KUKA KRL program: EPS_2_251825_SA25_A_20260116064101.src

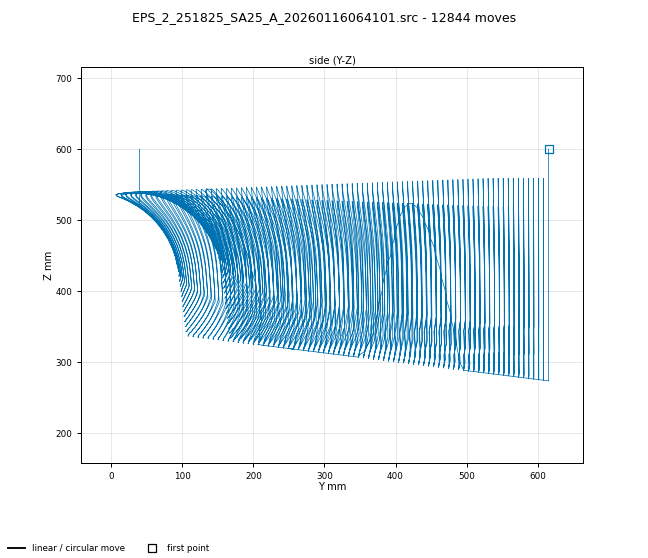
[picture p0: tool path of EPS_2_251825_SA25_A_20260116064101.src, 12844 of 12846 moves have a stored position in this frame; points joined in program order, loops and branches not executed]
&ACCESS RVP
&REL 4
&COMMENT QRS 19112012
&PARAM EDITMASK = *
DEF PART()
EXT BAS (BAS_COMMAND :IN,REAL :IN )
INT I
BAS (#INITMOV,0 )

;KUKA QRS Post kuka4.cps  Date:22-06-2017 !

File_ID=2984

QRS_PRE_INIT()

;Init var - Until changes are made in qrs_pre_init
Outlet_Square_prg=0
Inlet_1_Square_prg=0
Inlet_2_Square_prg=0
Inlet_3_Square_prg=0
Inlet_4_Square_prg=0
Inlet_5_Square_prg=0

Outlet_1={X 0.000, Y 535.490, Z 458.500, B 0.000, E1 0.000 }
Inlet_1={X 0.000, Y 538.340, Z 418.500, B 0.000, E1 170.000 }
Outlet_1_type=201
Inlet_1_type=201
;QRS#1=Sidecore dimensions
;QRS#2=200-8" PVC SDR 35
;QRS#3=200-8" PVC SDR 35
;QRS#4=
;QRS#5=
;QRS#6=
;QRS#7=
;QRS#8=
;QRS#9=12-08 PSX
;QRS#10=12-08 PSX
;QRS#11=
;QRS#12=
;QRS#13=
;QRS#14=
;QRS#15=
;QRS#16=1220x127x838 2,75'
;QRS#17=EPS Height
;QRS#18=559
;QRS#19=*
;QRS#20= UPDATED VERSION 22-06-2017
;QRS#21=*
Outlet_Square=0100
Inlet_1_Square=0100
Inlet_2_Square=0
Inlet_3_Square=0
Inlet_4_Square=0
Inlet_5_Square=0
Mill_Square=1
Outlet_Square_Prg=204
Inlet_1_Square_prg=204

QRS_INIT()

$ADVANCE=5

; T1
PTP {E1 173.614,E2 173.614}
PTP {X 0,Y 615.487,A -85,B 0,C 180,E1 173.614,E2 173.614,E3 0,E4 0,E5 0,E6 0}
QRS_SPEED_INIT()
LIN {X 0,Y 615.487,Z 600,A -85,B 0,C 180,E1 173.614,E2 173.614,E3 0,E4 0,E5 0,E6 0} C_VEL
LIN {X 0,Y 615.487,Z 283.875,A -85,B 0,C 180,E1 173.614,E2 173.614} C_VEL
LIN {X 0,Y 615.487,Z 275.693,A -85,B 0,C 180,E1 173.614,E2 173.614} C_VEL
LIN {X 0,Y 615.476,Z 273.693,A -85,B 0,C 180,E1 173.428,E2 173.428} C_VEL
LIN {X 0,Y 615.49,Z 273.68,A -85,B 0,C 180,E1 170.801,E2 170.801} C_VEL
LIN {X 0,Y 615.476,Z 273.688,A -85,B 0,C 180,E1 168.139,E2 168.139} C_VEL
LIN {X 0,Y 615.493,Z 273.698,A -85,B 0,C 180,E1 165.451,E2 165.451} C_VEL
LIN {X 0,Y 615.476,Z 273.685,A -85,B 0,C 180,E1 162.729,E2 162.729} C_VEL
LIN {X 0,Y 615.478,Z 273.686,A -85,B 0,C 180,E1 159.967,E2 159.967} C_VEL
LIN {X 0,Y 615.49,Z 273.698,A -85,B 0,C 180,E1 157.156,E2 157.156} C_VEL
LIN {X 0,Y 615.488,Z 273.681,A -85,B 0,C 180,E1 154.284,E2 154.284} C_VEL
LIN {X 0,Y 615.477,Z 273.689,A -85,B 0,C 180,E1 151.551,E2 151.551} C_VEL
LIN {X 0,Y 615.482,Z 273.7,A -85,B 0,C 180,E1 148.914,E2 148.914} C_VEL
LIN {X 0,Y 615.49,Z 273.68,A -85,B 0,C 180,E1 145.978,E2 145.978} C_VEL
LIN {X 0,Y 615.483,Z 273.694,A -85,B 0,C 180,E1 143.063,E2 143.063} C_VEL
LIN {X 0,Y 615.472,Z 273.69,A -85,B 0,C 180,E1 140.249,E2 140.249} C_VEL
LIN {X 0,Y 615.494,Z 273.679,A -85,B 0,C 180,E1 137.647,E2 137.647} C_VEL
LIN {X 0,Y 615.478,Z 273.692,A -85,B 0,C 180,E1 134.93,E2 134.93} C_VEL
LIN {X 0,Y 615.473,Z 273.692,A -85,B 0,C 180,E1 132.079,E2 132.079} C_VEL
LIN {X 0,Y 615.472,Z 273.686,A -85,B 0,C 180,E1 129.751,E2 129.751} C_VEL
LIN {X 0,Y 615.481,Z 273.685,A -85,B 0,C 180,E1 126.936,E2 126.936} C_VEL
LIN {X 0,Y 615.482,Z 273.696,A -85,B 0,C 180,E1 124.022,E2 124.022} C_VEL
LIN {X 0,Y 615.471,Z 273.691,A -85,B 0,C 180,E1 121.686,E2 121.686} C_VEL
LIN {X 0,Y 615.471,Z 273.686,A -85,B 0,C 180,E1 119.407,E2 119.407} C_VEL
LIN {X 0,Y 615.481,Z 273.787,A -85,B 0,C 180,E1 118.606,E2 118.606} C_VEL
LIN {X 0,Y 615.47,Z 289.754,A -85,B 0,C 180,E1 115.898,E2 115.898} C_VEL
LIN {X 0,Y 615.442,Z 304.793,A -85,B 0,C 180,E1 113.38,E2 113.38} C_VEL
LIN {X 0,Y 615.49,Z 308.179,A -85,B 0,C 180,E1 112.813,E2 112.813} C_VEL
LIN {X 0,Y 615.422,Z 414.922,A -85,B 0,C 180,E1 111.544,E2 111.544} C_VEL
LIN {X 0,Y 615.433,Z 427.931,A -85,B 0,C 180,E1 111.258,E2 111.258} C_VEL
LIN {X 0,Y 615.473,Z 440.076,A -85,B 0,C 180,E1 110.862,E2 110.862} C_VEL
LIN {X 0,Y 615.47,Z 451.61,A -85,B 0,C 180,E1 110.359,E2 110.359} C_VEL
LIN {X 0,Y 615.466,Z 462.135,A -85,B 0,C 180,E1 109.773,E2 109.773} C_VEL
LIN {X 0,Y 615.497,Z 473.243,A -85,B 0,C 180,E1 108.991,E2 108.991} C_VEL
LIN {X 0,Y 615.499,Z 481.455,A -85,B 0,C 180,E1 108.282,E2 108.282} C_VEL
LIN {X 0,Y 615.497,Z 489.66,A -85,B 0,C 180,E1 107.442,E2 107.442} C_VEL
LIN {X 0,Y 615.496,Z 497.619,A -85,B 0,C 180,E1 106.433,E2 106.433} C_VEL
LIN {X 0,Y 615.495,Z 503.176,A -85,B 0,C 180,E1 105.565,E2 105.565} C_VEL
LIN {X 0,Y 615.497,Z 508.401,A -85,B 0,C 180,E1 104.549,E2 104.549} C_VEL
LIN {X 0,Y 615.496,Z 512.408,A -85,B 0,C 180,E1 103.537,E2 103.537} C_VEL
LIN {X 0,Y 615.494,Z 515.337,A -85,B 0,C 180,E1 102.53,E2 102.53} C_VEL
LIN {X 0,Y 615.496,Z 516.703,A -85,B 0,C 180,E1 101.861,E2 101.861} C_VEL
LIN {X 0,Y 615.496,Z 518.232,A -85,B 0,C 180,E1 100.527,E2 100.527} C_VEL
LIN {X 0,Y 615.496,Z 518.372,A -85,B 0,C 180,E1 99.862,E2 99.862} C_VEL
LIN {X 0,Y 615.496,Z 517.451,A -85,B 0,C 180,E1 98.537,E2 98.537} C_VEL
LIN {X 0,Y 615.494,Z 516.408,A -85,B 0,C 180,E1 97.876,E2 97.876} C_VEL
LIN {X 0,Y 615.495,Z 513.082,A -85,B 0,C 180,E1 96.583,E2 96.583} C_VEL
LIN {X 0,Y 615.496,Z 509.298,A -85,B 0,C 180,E1 95.57,E2 95.57} C_VEL
LIN {X 0,Y 615.498,Z 504.497,A -85,B 0,C 180,E1 94.585,E2 94.585} C_VEL
LIN {X 0,Y 615.491,Z 498.461,A -85,B 0,C 180,E1 93.601,E2 93.601} C_VEL
LIN {X 0,Y 615.498,Z 490.972,A -85,B 0,C 180,E1 92.618,E2 92.618} C_VEL
LIN {X 0,Y 615.497,Z 483.209,A -85,B 0,C 180,E1 91.8,E2 91.8} C_VEL
LIN {X 0,Y 615.5,Z 475.088,A -85,B 0,C 180,E1 91.064,E2 91.064} C_VEL
LIN {X 0,Y 615.493,Z 465.046,A -85,B 0,C 180,E1 90.327,E2 90.327} C_VEL
LIN {X 0,Y 615.486,Z 453.961,A -85,B 0,C 180,E1 89.673,E2 89.673} C_VEL
LIN {X 0,Y 615.491,Z 443.467,A -85,B 0,C 180,E1 89.183,E2 89.183} C_VEL
LIN {X 0,Y 615.461,Z 430.84,A -85,B 0,C 180,E1 88.733,E2 88.733} C_VEL
LIN {X 0,Y 615.462,Z 418.151,A -85,B 0,C 180,E1 88.426,E2 88.426} C_VEL
LIN {X 0,Y 615.475,Z 400.264,A -85,B 0,C 180,E1 88.18,E2 88.18} C_VEL
LIN {X 0,Y 615.467,Z 308.178,A -85,B 0,C 180,E1 87.096,E2 87.096} C_VEL
LIN {X 0,Y 615.429,Z 294.206,A -85,B 0,C 180,E1 84.759,E2 84.759} C_VEL
LIN {X 0,Y 615.432,Z 280.557,A -85,B 0,C 180,E1 82.454,E2 82.454} C_VEL
LIN {X 0,Y 615.438,Z 273.696,A -85,B 0,C 180,E1 81.256,E2 81.256} C_VEL
LIN {X 0,Y 615.418,Z 273.696,A -85,B 0,C 180,E1 78.806,E2 78.806} C_VEL
LIN {X 0,Y 615.42,Z 273.696,A -85,B 0,C 180,E1 76.798,E2 76.798} C_VEL
LIN {X 0,Y 615.42,Z 273.696,A -85,B 0,C 180,E1 74.773,E2 74.773} C_VEL
LIN {X 0,Y 615.424,Z 273.695,A -85,B 0,C 180,E1 72.728,E2 72.728} C_VEL
LIN {X 0,Y 615.424,Z 273.695,A -85,B 0,C 180,E1 70.661,E2 70.661} C_VEL
LIN {X 0,Y 615.425,Z 273.695,A -85,B 0,C 180,E1 68.567,E2 68.567} C_VEL
LIN {X 0,Y 615.423,Z 273.695,A -85,B 0,C 180,E1 66.442,E2 66.442} C_VEL
LIN {X 0,Y 615.425,Z 273.695,A -85,B 0,C 180,E1 64.282,E2 64.282} C_VEL
LIN {X 0,Y 615.428,Z 273.696,A -85,B 0,C 180,E1 62.083,E2 62.083} C_VEL
LIN {X 0,Y 615.492,Z 273.695,A -85,B 0,C 180,E1 59.081,E2 59.081} C_VEL
LIN {X 0,Y 615.448,Z 273.691,A -85,B 0,C 180,E1 56.471,E2 56.471} C_VEL
LIN {X 0,Y 615.434,Z 273.693,A -85,B 0,C 180,E1 54.173,E2 54.173} C_VEL
LIN {X 0,Y 615.432,Z 273.694,A -85,B 0,C 180,E1 51.929,E2 51.929} C_VEL
LIN {X 0,Y 615.452,Z 273.697,A -85,B 0,C 180,E1 49.392,E2 49.392} C_VEL
LIN {X 0,Y 615.497,Z 273.694,A -85,B 0,C 180,E1 46.757,E2 46.757} C_VEL
LIN {X 0,Y 615.447,Z 273.69,A -85,B 0,C 180,E1 43.995,E2 43.995} C_VEL
LIN {X 0,Y 615.439,Z 273.694,A -85,B 0,C 180,E1 41.478,E2 41.478} C_VEL
LIN {X 0,Y 615.473,Z 273.699,A -85,B 0,C 180,E1 38.905,E2 38.905} C_VEL
LIN {X 0,Y 615.495,Z 273.692,A -85,B 0,C 180,E1 36.424,E2 36.424} C_VEL
LIN {X 0,Y 615.485,Z 273.685,A -85,B 0,C 180,E1 34.022,E2 34.022} C_VEL
LIN {X 0,Y 615.458,Z 273.688,A -85,B 0,C 180,E1 31.687,E2 31.687} C_VEL
LIN {X 0,Y 615.446,Z 273.69,A -85,B 0,C 180,E1 29.408,E2 29.408} C_VEL
LIN {X 0,Y 615.446,Z 273.693,A -85,B 0,C 180,E1 27.04,E2 27.04} C_VEL
LIN {X 0,Y 615.492,Z 273.699,A -85,B 0,C 180,E1 24.272,E2 24.272} C_VEL
LIN {X 0,Y 615.467,Z 273.686,A -85,B 0,C 180,E1 21.433,E2 21.433} C_VEL
LIN {X 0,Y 615.466,Z 273.686,A -85,B 0,C 180,E1 19.339,E2 19.339} C_VEL
LIN {X 0,Y 615.463,Z 273.686,A -85,B 0,C 180,E1 17.271,E2 17.271} C_VEL
LIN {X 0,Y 615.469,Z 273.685,A -85,B 0,C 180,E1 15.226,E2 15.226} C_VEL
LIN {X 0,Y 615.473,Z 273.685,A -85,B 0,C 180,E1 13.201,E2 13.201} C_VEL
LIN {X 0,Y 615.454,Z 273.692,A -85,B 0,C 180,E1 10.527,E2 10.527} C_VEL
LIN {X 0,Y 615.487,Z 273.702,A -85,B 0,C 180,E1 7.876,E2 7.876} C_VEL
LIN {X 0,Y 615.491,Z 273.684,A -85,B 0,C 180,E1 5.241,E2 5.241} C_VEL
LIN {X 0,Y 615.46,Z 273.687,A -85,B 0,C 180,E1 2.618,E2 2.618} C_VEL
LIN {X 0,Y 615.469,Z 273.695,A -85,B 0,C 180,E1 0,E2 0} C_VEL
LIN {X 0,Y 615.489,Z 273.693,A -85,B 0,C 180,E1 -2.618,E2 -2.618} C_VEL
LIN {X 0,Y 615.487,Z 273.682,A -85,B 0,C 180,E1 -5.241,E2 -5.241} C_VEL
LIN {X 0,Y 615.461,Z 273.689,A -85,B 0,C 180,E1 -7.876,E2 -7.876} C_VEL
LIN {X 0,Y 615.485,Z 273.701,A -85,B 0,C 180,E1 -10.527,E2 -10.527} C_VEL
LIN {X 0,Y 615.487,Z 273.686,A -85,B 0,C 180,E1 -13.201,E2 -13.201} C_VEL
LIN {X 0,Y 615.469,Z 273.685,A -85,B 0,C 180,E1 -15.906,E2 -15.906} C_VEL
LIN {X 0,Y 615.48,Z 273.698,A -85,B 0,C 180,E1 -18.646,E2 -18.646} C_VEL
LIN {X 0,Y 615.48,Z 273.687,A -85,B 0,C 180,E1 -21.432,E2 -21.432} C_VEL
LIN {X 0,Y 615.468,Z 273.687,A -85,B 0,C 180,E1 -24.273,E2 -24.273} C_VEL
LIN {X 0,Y 615.496,Z 273.701,A -85,B 0,C 180,E1 -27.049,E2 -27.049} C_VEL
LIN {X 0,Y 615.487,Z 273.683,A -85,B 0,C 180,E1 -29.797,E2 -29.797} C_VEL
LIN {X 0,Y 615.473,Z 273.686,A -85,B 0,C 180,E1 -32.459,E2 -32.459} C_VEL
LIN {X 0,Y 615.472,Z 273.691,A -85,B 0,C 180,E1 -34.816,E2 -34.816} C_VEL
LIN {X 0,Y 615.487,Z 273.7,A -85,B 0,C 180,E1 -37.242,E2 -37.242} C_VEL
LIN {X 0,Y 615.481,Z 273.684,A -85,B 0,C 180,E1 -40.09,E2 -40.09} C_VEL
LIN {X 0,Y 615.494,Z 273.679,A -85,B 0,C 180,E1 -42.353,E2 -42.353} C_VEL
LIN {X 0,Y 615.475,Z 273.69,A -85,B 0,C 180,E1 -45.07,E2 -45.07} C_VEL
LIN {X 0,Y 615.478,Z 273.693,A -85,B 0,C 180,E1 -47.921,E2 -47.921} C_VEL
LIN {X 0,Y 615.475,Z 273.687,A -85,B 0,C 180,E1 -50.25,E2 -50.25} C_VEL
LIN {X 0,Y 615.481,Z 273.685,A -85,B 0,C 180,E1 -53.065,E2 -53.065} C_VEL
LIN {X 0,Y 615.485,Z 273.697,A -85,B 0,C 180,E1 -55.979,E2 -55.979} C_VEL
LIN {X 0,Y 615.472,Z 273.691,A -85,B 0,C 180,E1 -58.315,E2 -58.315} C_VEL
LIN {X 0,Y 615.472,Z 273.687,A -85,B 0,C 180,E1 -60.594,E2 -60.594} C_VEL
LIN {X 0,Y 615.487,Z 273.681,A -85,B 0,C 180,E1 -62.956,E2 -62.956} C_VEL
LIN {X 0,Y 615.481,Z 273.692,A -85,B 0,C 180,E1 -65.728,E2 -65.728} C_VEL
LIN {X 0,Y 615.487,Z 273.756,A -85,B 0,C 180,E1 -67.438,E2 -67.438} C_VEL
LIN {X 0,Y 615.455,Z 293.696,A -85,B 0,C 180,E1 -70.141,E2 -70.141} C_VEL
LIN {X 0,Y 615.472,Z 313.082,A -85,B 0,C 180,E1 -72.73,E2 -72.73} C_VEL
LIN {X 0,Y 615.493,Z 334.92,A -85,B 0,C 180,E1 -75.607,E2 -75.607} C_VEL
LIN {X 0,Y 615.471,Z 346.472,A -85,B 0,C 180,E1 -77.114,E2 -77.114} C_VEL
LIN {X 0,Y 615.457,Z 454.866,A -85,B 0,C 180,E1 -78.411,E2 -78.411} C_VEL
LIN {X 0,Y 615.456,Z 467.368,A -85,B 0,C 180,E1 -78.682,E2 -78.682} C_VEL
LIN {X 0,Y 615.483,Z 480.688,A -85,B 0,C 180,E1 -79.116,E2 -79.116} C_VEL
LIN {X 0,Y 615.492,Z 492.486,A -85,B 0,C 180,E1 -79.64,E2 -79.64} C_VEL
LIN {X 0,Y 615.483,Z 504.003,A -85,B 0,C 180,E1 -80.304,E2 -80.304} C_VEL
LIN {X 0,Y 615.499,Z 514.347,A -85,B 0,C 180,E1 -81.05,E2 -81.05} C_VEL
LIN {X 0,Y 615.497,Z 522.696,A -85,B 0,C 180,E1 -81.795,E2 -81.795} C_VEL
LIN {X 0,Y 615.498,Z 530.61,A -85,B 0,C 180,E1 -82.62,E2 -82.62} C_VEL
LIN {X 0,Y 615.491,Z 538.207,A -85,B 0,C 180,E1 -83.608,E2 -83.608} C_VEL
LIN {X 0,Y 615.498,Z 545.207,A -85,B 0,C 180,E1 -84.759,E2 -84.759} C_VEL
LIN {X 0,Y 615.493,Z 549.853,A -85,B 0,C 180,E1 -85.744,E2 -85.744} C_VEL
LIN {X 0,Y 615.494,Z 553.4,A -85,B 0,C 180,E1 -86.727,E2 -86.727} C_VEL
LIN {X 0,Y 615.497,Z 555.234,A -85,B 0,C 180,E1 -87.383,E2 -87.383} C_VEL
LIN {X 0,Y 615.497,Z 556.609,A -85,B 0,C 180,E1 -88.037,E2 -88.037} C_VEL
LIN {X 0,Y 615.496,Z 558.174,A -85,B 0,C 180,E1 -89.346,E2 -89.346} C_VEL
LIN {X 0,Y 615.494,Z 558.389,A -85,B 0,C 180,E1 -90,E2 -90} C_VEL
LIN {X 0,Y 615.495,Z 557.58,A -85,B 0,C 180,E1 -91.309,E2 -91.309} C_VEL
LIN {X 0,Y 615.497,Z 556.608,A -85,B 0,C 180,E1 -91.963,E2 -91.963} C_VEL
LIN {X 0,Y 615.497,Z 555.232,A -85,B 0,C 180,E1 -92.618,E2 -92.618} C_VEL
LIN {X 0,Y 615.496,Z 552.348,A -85,B 0,C 180,E1 -93.601,E2 -93.601} C_VEL
LIN {X 0,Y 615.498,Z 548.44,A -85,B 0,C 180,E1 -94.585,E2 -94.585} C_VEL
LIN {X 0,Y 615.499,Z 543.403,A -85,B 0,C 180,E1 -95.57,E2 -95.57} C_VEL
LIN {X 0,Y 615.49,Z 536.913,A -85,B 0,C 180,E1 -96.578,E2 -96.578} C_VEL
LIN {X 0,Y 615.497,Z 529.131,A -85,B 0,C 180,E1 -97.546,E2 -97.546} C_VEL
LIN {X 0,Y 615.498,Z 519.255,A -85,B 0,C 180,E1 -98.537,E2 -98.537} C_VEL
LIN {X 0,Y 615.495,Z 508.863,A -85,B 0,C 180,E1 -99.365,E2 -99.365} C_VEL
LIN {X 0,Y 615.482,Z 498.572,A -85,B 0,C 180,E1 -100.029,E2 -100.029} C_VEL
LIN {X 0,Y 615.495,Z 487.133,A -85,B 0,C 180,E1 -100.616,E2 -100.616} C_VEL
LIN {X 0,Y 615.467,Z 475.354,A -85,B 0,C 180,E1 -101.078,E2 -101.078} C_VEL
LIN {X 0,Y 615.455,Z 462.238,A -85,B 0,C 180,E1 -101.444,E2 -101.444} C_VEL
LIN {X 0,Y 615.461,Z 448.933,A -85,B 0,C 180,E1 -101.674,E2 -101.674} C_VEL
LIN {X 0,Y 615.471,Z 346.467,A -85,B 0,C 180,E1 -102.887,E2 -102.887} C_VEL
LIN {X 0,Y 615.455,Z 325.989,A -85,B 0,C 180,E1 -105.566,E2 -105.566} C_VEL
LIN {X 0,Y 615.481,Z 305.474,A -85,B 0,C 180,E1 -108.281,E2 -108.281} C_VEL
LIN {X 0,Y 615.468,Z 283.343,A -85,B 0,C 180,E1 -111.257,E2 -111.257} C_VEL
LIN {X 0,Y 615.489,Z 273.682,A -85,B 0,C 180,E1 -112.594,E2 -112.594} C_VEL
LIN {X 0,Y 615.485,Z 273.681,A -85,B 0,C 180,E1 -114.992,E2 -114.992} C_VEL
LIN {X 0,Y 615.482,Z 273.698,A -85,B 0,C 180,E1 -117.915,E2 -117.915} C_VEL
LIN {X 0,Y 615.486,Z 273.682,A -85,B 0,C 180,E1 -120.92,E2 -120.92} C_VEL
LIN {X 0,Y 615.471,Z 273.686,A -85,B 0,C 180,E1 -123.531,E2 -123.531} C_VEL
LIN {X 0,Y 615.486,Z 273.699,A -85,B 0,C 180,E1 -126.425,E2 -126.425} C_VEL
LIN {X 0,Y 615.481,Z 273.685,A -85,B 0,C 180,E1 -129.061,E2 -129.061} C_VEL
LIN {X 0,Y 615.491,Z 273.68,A -85,B 0,C 180,E1 -131.473,E2 -131.473} C_VEL
LIN {X 0,Y 615.469,Z 273.692,A -85,B 0,C 180,E1 -134.151,E2 -134.151} C_VEL
LIN {X 0,Y 615.482,Z 273.693,A -85,B 0,C 180,E1 -136.953,E2 -136.953} C_VEL
LIN {X 0,Y 615.483,Z 273.684,A -85,B 0,C 180,E1 -139.393,E2 -139.393} C_VEL
LIN {X 0,Y 615.479,Z 273.683,A -85,B 0,C 180,E1 -141.989,E2 -141.989} C_VEL
LIN {X 0,Y 615.471,Z 273.69,A -85,B 0,C 180,E1 -144.383,E2 -144.383} C_VEL
LIN {X 0,Y 615.477,Z 273.697,A -85,B 0,C 180,E1 -146.763,E2 -146.763} C_VEL
LIN {X 0,Y 615.487,Z 273.701,A -85,B 0,C 180,E1 -149.08,E2 -149.08} C_VEL
LIN {X 0,Y 615.484,Z 273.681,A -85,B 0,C 180,E1 -152.085,E2 -152.085} C_VEL
LIN {X 0,Y 615.482,Z 273.696,A -85,B 0,C 180,E1 -155.008,E2 -155.008} C_VEL
LIN {X 0,Y 615.478,Z 273.687,A -85,B 0,C 180,E1 -157.863,E2 -157.863} C_VEL
LIN {X 0,Y 615.477,Z 273.684,A -85,B 0,C 180,E1 -160.662,E2 -160.662} C_VEL
LIN {X 0,Y 615.486,Z 273.7,A -85,B 0,C 180,E1 -163.568,E2 -163.568} C_VEL
LIN {X 0,Y 615.476,Z 273.688,A -85,B 0,C 180,E1 -166.125,E2 -166.125} C_VEL
LIN {X 0,Y 615.485,Z 273.681,A -85,B 0,C 180,E1 -168.807,E2 -168.807} C_VEL
LIN {X 0,Y 615.479,Z 273.694,A -85,B 0,C 180,E1 -171.463,E2 -171.463} C_VEL
LIN {X 0,Y 615.48,Z 273.694,A -85,B 0,C 180,E1 -174.101,E2 -174.101} C_VEL
LIN {X 0,Y 615.487,Z 273.681,A -85,B 0,C 180,E1 -176.727,E2 -176.727} C_VEL
LIN {X 0,Y 615.474,Z 273.686,A -85,B 0,C 180,E1 -179.346,E2 -179.346} C_VEL
LIN {X 0,Y 615.49,Z 273.698,A -85,B 0,C 180,E1 -181.963,E2 -181.963} C_VEL
LIN {X 0,Y 615.476,Z 273.69,A -85,B 0,C 180,E1 -184.585,E2 -184.585} C_VEL
LIN {X 0,Y 615.476,Z 273.693,A -85,B 0,C 180,E1 -186.572,E2 -186.572} C_VEL
LIN {X 0,Y 614.808,Z 273.83,A -85,B 0,C 180,E1 -187.118,E2 -187.118} C_VEL
LIN {X 0,Y 611.982,Z 274.253,A -85,B 0,C 180,E1 -188.004,E2 -188.004} C_VEL
LIN {X 0,Y 609.591,Z 274.559,A -85,B 0,C 180,E1 -188.717,E2 -188.717} C_VEL
LIN {X 0,Y 608.551,Z 274.675,A -85,B 0,C 180,E1 -189.267,E2 -189.267} C_VEL
LIN {X 0,Y 608.459,Z 274.686,A -85,B 0,C 180,E1 -189.453,E2 -189.453} C_VEL
LIN {X 0,Y 608.454,Z 274.691,A -85,B 0,C 180,E1 -192,E2 -192} C_VEL
LIN {X 0,Y 608.477,Z 274.69,A -85,B 0,C 180,E1 -194.72,E2 -194.72} C_VEL
LIN {X 0,Y 608.444,Z 274.687,A -85,B 0,C 180,E1 -197.477,E2 -197.477} C_VEL
LIN {X 0,Y 608.445,Z 274.687,A -85,B 0,C 180,E1 -199.571,E2 -199.571} C_VEL
LIN {X 0,Y 608.474,Z 274.689,A -85,B 0,C 180,E1 -202.405,E2 -202.405} C_VEL
LIN {X 0,Y 608.448,Z 274.694,A -85,B 0,C 180,E1 -204.571,E2 -204.571} C_VEL
LIN {X 0,Y 608.473,Z 274.689,A -85,B 0,C 180,E1 -207.207,E2 -207.207} C_VEL
LIN {X 0,Y 608.466,Z 274.685,A -85,B 0,C 180,E1 -209.972,E2 -209.972} C_VEL
LIN {X 0,Y 608.452,Z 274.695,A -85,B 0,C 180,E1 -212.88,E2 -212.88} C_VEL
LIN {X 0,Y 608.434,Z 274.697,A -85,B 0,C 180,E1 -215.278,E2 -215.278} C_VEL
LIN {X 0,Y 608.467,Z 274.687,A -85,B 0,C 180,E1 -217.746,E2 -217.746} C_VEL
LIN {X 0,Y 608.446,Z 274.687,A -85,B 0,C 180,E1 -220.329,E2 -220.329} C_VEL
LIN {X 0,Y 608.477,Z 274.694,A -85,B 0,C 180,E1 -223.31,E2 -223.31} C_VEL
LIN {X 0,Y 608.459,Z 274.687,A -85,B 0,C 180,E1 -226.13,E2 -226.13} C_VEL
LIN {X 0,Y 608.454,Z 274.687,A -85,B 0,C 180,E1 -228.824,E2 -228.824} C_VEL
LIN {X 0,Y 608.46,Z 274.695,A -85,B 0,C 180,E1 -231.761,E2 -231.761} C_VEL
LIN {X 0,Y 608.444,Z 274.694,A -85,B 0,C 180,E1 -233.955,E2 -233.955} C_VEL
LIN {X 0,Y 608.442,Z 274.69,A -85,B 0,C 180,E1 -236.328,E2 -236.328} C_VEL
LIN {X 0,Y 608.445,Z 274.688,A -85,B 0,C 180,E1 -238.733,E2 -238.733} C_VEL
LIN {X 0,Y 608.483,Z 274.798,A -85,B 0,C 180,E1 -241.335,E2 -241.335} C_VEL
LIN {X 0,Y 608.46,Z 290.176,A -85,B 0,C 180,E1 -243.965,E2 -243.965} C_VEL
LIN {X 0,Y 608.433,Z 305.278,A -85,B 0,C 180,E1 -246.515,E2 -246.515} C_VEL
LIN {X 0,Y 608.493,Z 308.602,A -85,B 0,C 180,E1 -247.046,E2 -247.046} C_VEL
LIN {X 0,Y 608.485,Z 415.533,A -85,B 0,C 180,E1 -248.331,E2 -248.331} C_VEL
LIN {X 0,Y 608.487,Z 429.172,A -85,B 0,C 180,E1 -248.643,E2 -248.643} C_VEL
LIN {X 0,Y 608.519,Z 441.754,A -85,B 0,C 180,E1 -249.07,E2 -249.07} C_VEL
LIN {X 0,Y 608.473,Z 453.212,A -85,B 0,C 180,E1 -249.594,E2 -249.594} C_VEL
LIN {X 0,Y 608.477,Z 464.479,A -85,B 0,C 180,E1 -250.254,E2 -250.254} C_VEL
LIN {X 0,Y 608.473,Z 475.262,A -85,B 0,C 180,E1 -251.043,E2 -251.043} C_VEL
LIN {X 0,Y 608.465,Z 483.865,A -85,B 0,C 180,E1 -251.829,E2 -251.829} C_VEL
LIN {X 0,Y 608.471,Z 490.475,A -85,B 0,C 180,E1 -252.524,E2 -252.524} C_VEL
LIN {X 0,Y 608.468,Z 497.893,A -85,B 0,C 180,E1 -253.471,E2 -253.471} C_VEL
LIN {X 0,Y 608.431,Z 504.862,A -85,B 0,C 180,E1 -254.593,E2 -254.593} C_VEL
LIN {X 0,Y 608.431,Z 509.862,A -85,B 0,C 180,E1 -255.62,E2 -255.62} C_VEL
LIN {X 0,Y 608.444,Z 513.665,A -85,B 0,C 180,E1 -256.643,E2 -256.643} C_VEL
LIN {X 0,Y 608.42,Z 515.611,A -85,B 0,C 180,E1 -257.322,E2 -257.322} C_VEL
LIN {X 0,Y 608.44,Z 517.102,A -85,B 0,C 180,E1 -258,E2 -258} C_VEL
LIN {X 0,Y 608.437,Z 518.76,A -85,B 0,C 180,E1 -259.349,E2 -259.349} C_VEL
LIN {X 0,Y 608.432,Z 518.999,A -85,B 0,C 180,E1 -260.022,E2 -260.022} C_VEL
LIN {X 0,Y 608.42,Z 518.793,A -85,B 0,C 180,E1 -260.693,E2 -260.693} C_VEL
LIN {X 0,Y 608.419,Z 517.199,A -85,B 0,C 180,E1 -262.032,E2 -262.032} C_VEL
LIN {X 0,Y 608.423,Z 515.792,A -85,B 0,C 180,E1 -262.7,E2 -262.7} C_VEL
LIN {X 0,Y 608.452,Z 513.088,A -85,B 0,C 180,E1 -263.628,E2 -263.628} C_VEL
LIN {X 0,Y 608.44,Z 508.886,A -85,B 0,C 180,E1 -264.698,E2 -264.698} C_VEL
LIN {X 0,Y 608.438,Z 502.792,A -85,B 0,C 180,E1 -265.86,E2 -265.86} C_VEL
LIN {X 0,Y 608.456,Z 496.159,A -85,B 0,C 180,E1 -266.855,E2 -266.855} C_VEL
LIN {X 0,Y 608.454,Z 487.961,A -85,B 0,C 180,E1 -267.848,E2 -267.848} C_VEL
LIN {X 0,Y 608.479,Z 477.675,A -85,B 0,C 180,E1 -268.841,E2 -268.841} C_VEL
LIN {X 0,Y 608.479,Z 467,A -85,B 0,C 180,E1 -269.669,E2 -269.669} C_VEL
LIN {X 0,Y 608.499,Z 456.28,A -85,B 0,C 180,E1 -270.331,E2 -270.331} C_VEL
LIN {X 0,Y 608.527,Z 444.369,A -85,B 0,C 180,E1 -270.91,E2 -270.91} C_VEL
LIN {X 0,Y 608.518,Z 431.984,A -85,B 0,C 180,E1 -271.365,E2 -271.365} C_VEL
LIN {X 0,Y 608.508,Z 418.923,A -85,B 0,C 180,E1 -271.696,E2 -271.696} C_VEL
LIN {X 0,Y 608.532,Z 403.179,A -85,B 0,C 180,E1 -271.923,E2 -271.923} C_VEL
LIN {X 0,Y 608.49,Z 308.827,A -85,B 0,C 180,E1 -273.041,E2 -273.041} C_VEL
LIN {X 0,Y 608.448,Z 308.334,A -85,B 0,C 180,E1 -273.062,E2 -273.062} C_VEL
LIN {X 0,Y 608.413,Z 293.074,A -85,B 0,C 180,E1 -275.634,E2 -275.634} C_VEL
LIN {X 0,Y 608.494,Z 277.439,A -85,B 0,C 180,E1 -278.3,E2 -278.3} C_VEL
LIN {X 0,Y 608.417,Z 274.693,A -85,B 0,C 180,E1 -278.803,E2 -278.803} C_VEL
LIN {X 0,Y 608.403,Z 274.693,A -85,B 0,C 180,E1 -281.325,E2 -281.325} C_VEL
LIN {X 0,Y 608.407,Z 274.692,A -85,B 0,C 180,E1 -283.357,E2 -283.357} C_VEL
LIN {X 0,Y 608.416,Z 274.691,A -85,B 0,C 180,E1 -285.407,E2 -285.407} C_VEL
LIN {X 0,Y 608.402,Z 274.693,A -85,B 0,C 180,E1 -287.477,E2 -287.477} C_VEL
LIN {X 0,Y 608.402,Z 274.693,A -85,B 0,C 180,E1 -289.572,E2 -289.572} C_VEL
LIN {X 0,Y 608.422,Z 274.691,A -85,B 0,C 180,E1 -291.693,E2 -291.693} C_VEL
LIN {X 0,Y 608.436,Z 274.7,A -85,B 0,C 180,E1 -294.571,E2 -294.571} C_VEL
LIN {X 0,Y 608.416,Z 274.691,A -85,B 0,C 180,E1 -297.519,E2 -297.519} C_VEL
LIN {X 0,Y 608.4,Z 274.694,A -85,B 0,C 180,E1 -299.96,E2 -299.96} C_VEL
LIN {X 0,Y 608.437,Z 274.695,A -85,B 0,C 180,E1 -302.519,E2 -302.519} C_VEL
LIN {X 0,Y 608.424,Z 274.694,A -85,B 0,C 180,E1 -305.278,E2 -305.278} C_VEL
LIN {X 0,Y 608.437,Z 274.689,A -85,B 0,C 180,E1 -307.748,E2 -307.748} C_VEL
LIN {X 0,Y 608.427,Z 274.691,A -85,B 0,C 180,E1 -310.326,E2 -310.326} C_VEL
LIN {X 0,Y 608.445,Z 274.697,A -85,B 0,C 180,E1 -312.959,E2 -312.959} C_VEL
LIN {X 0,Y 608.434,Z 274.691,A -85,B 0,C 180,E1 -315.737,E2 -315.737} C_VEL
LIN {X 0,Y 608.441,Z 274.689,A -85,B 0,C 180,E1 -317.937,E2 -317.937} C_VEL
LIN {X 0,Y 608.418,Z 274.693,A -85,B 0,C 180,E1 -320.707,E2 -320.707} C_VEL
LIN {X 0,Y 608.437,Z 274.695,A -85,B 0,C 180,E1 -323.084,E2 -323.084} C_VEL
LIN {X 0,Y 608.467,Z 274.694,A -85,B 0,C 180,E1 -325.531,E2 -325.531} C_VEL
LIN {X 0,Y 608.462,Z 274.689,A -85,B 0,C 180,E1 -327.905,E2 -327.905} C_VEL
LIN {X 0,Y 608.459,Z 274.687,A -85,B 0,C 180,E1 -330.22,E2 -330.22} C_VEL
LIN {X 0,Y 608.423,Z 274.69,A -85,B 0,C 180,E1 -332.801,E2 -332.801} C_VEL
LIN {X 0,Y 608.44,Z 274.695,A -85,B 0,C 180,E1 -335.428,E2 -335.428} C_VEL
LIN {X 0,Y 608.459,Z 274.688,A -85,B 0,C 180,E1 -338.308,E2 -338.308} C_VEL
LIN {X 0,Y 608.435,Z 274.69,A -85,B 0,C 180,E1 -341.13,E2 -341.13} C_VEL
LIN {X 0,Y 608.477,Z 274.695,A -85,B 0,C 180,E1 -343.907,E2 -343.907} C_VEL
LIN {X 0,Y 608.455,Z 274.687,A -85,B 0,C 180,E1 -346.643,E2 -346.643} C_VEL
LIN {X 0,Y 608.435,Z 274.69,A -85,B 0,C 180,E1 -349.35,E2 -349.35} C_VEL
LIN {X 0,Y 608.472,Z 274.694,A -85,B 0,C 180,E1 -352.033,E2 -352.033} C_VEL
LIN {X 0,Y 608.47,Z 274.687,A -85,B 0,C 180,E1 -354.698,E2 -354.698} C_VEL
LIN {X 0,Y 608.454,Z 274.686,A -85,B 0,C 180,E1 -357.352,E2 -357.352} C_VEL
LIN {X 0,Y 608.46,Z 274.691,A -85,B 0,C 180,E1 -360,E2 -360} C_VEL
LIN {X 0,Y 608.479,Z 274.69,A -85,B 0,C 180,E1 -362.648,E2 -362.648} C_VEL
LIN {X 0,Y 608.463,Z 274.685,A -85,B 0,C 180,E1 -365.302,E2 -365.302} C_VEL
LIN {X 0,Y 608.458,Z 274.688,A -85,B 0,C 180,E1 -367.967,E2 -367.967} C_VEL
LIN {X 0,Y 608.464,Z 274.696,A -85,B 0,C 180,E1 -370.65,E2 -370.65} C_VEL
LIN {X 0,Y 608.459,Z 274.687,A -85,B 0,C 180,E1 -373.357,E2 -373.357} C_VEL
LIN {X 0,Y 608.445,Z 274.689,A -85,B 0,C 180,E1 -376.094,E2 -376.094} C_VEL
LIN {X 0,Y 608.45,Z 274.698,A -85,B 0,C 180,E1 -378.87,E2 -378.87} C_VEL
LIN {X 0,Y 608.459,Z 274.686,A -85,B 0,C 180,E1 -381.692,E2 -381.692} C_VEL
LIN {X 0,Y 608.446,Z 274.692,A -85,B 0,C 180,E1 -384.572,E2 -384.572} C_VEL
LIN {X 0,Y 608.482,Z 274.691,A -85,B 0,C 180,E1 -387.21,E2 -387.21} C_VEL
LIN {X 0,Y 608.467,Z 274.685,A -85,B 0,C 180,E1 -389.973,E2 -389.973} C_VEL
LIN {X 0,Y 608.45,Z 274.688,A -85,B 0,C 180,E1 -392.522,E2 -392.522} C_VEL
LIN {X 0,Y 608.438,Z 274.693,A -85,B 0,C 180,E1 -394.906,E2 -394.906} C_VEL
LIN {X 0,Y 608.474,Z 274.693,A -85,B 0,C 180,E1 -397.16,E2 -397.16} C_VEL
LIN {X 0,Y 608.466,Z 274.695,A -85,B 0,C 180,E1 -399.44,E2 -399.44} C_VEL
LIN {X 0,Y 608.465,Z 274.685,A -85,B 0,C 180,E1 -402.336,E2 -402.336} C_VEL
LIN {X 0,Y 608.445,Z 274.693,A -85,B 0,C 180,E1 -405.204,E2 -405.204} C_VEL
LIN {X 0,Y 608.458,Z 274.691,A -85,B 0,C 180,E1 -407.94,E2 -407.94} C_VEL
LIN {X 0,Y 608.44,Z 274.688,A -85,B 0,C 180,E1 -410.706,E2 -410.706} C_VEL
LIN {X 0,Y 608.452,Z 274.688,A -85,B 0,C 180,E1 -413.086,E2 -413.086} C_VEL
LIN {X 0,Y 608.465,Z 274.691,A -85,B 0,C 180,E1 -415.531,E2 -415.531} C_VEL
LIN {X 0,Y 608.463,Z 274.696,A -85,B 0,C 180,E1 -417.906,E2 -417.906} C_VEL
LIN {X 0,Y 608.463,Z 274.691,A -85,B 0,C 180,E1 -420.221,E2 -420.221} C_VEL
LIN {X 0,Y 608.474,Z 274.684,A -85,B 0,C 180,E1 -422.794,E2 -422.794} C_VEL
LIN {X 0,Y 608.451,Z 274.688,A -85,B 0,C 180,E1 -425.43,E2 -425.43} C_VEL
LIN {X 0,Y 608.506,Z 274.826,A -85,B 0,C 180,E1 -427.313,E2 -427.313} C_VEL
LIN {X 0,Y 608.524,Z 292.412,A -85,B 0,C 180,E1 -429.729,E2 -429.729} C_VEL
LIN {X 0,Y 608.51,Z 311.829,A -85,B 0,C 180,E1 -432.352,E2 -432.352} C_VEL
LIN {X 0,Y 608.496,Z 332.54,A -85,B 0,C 180,E1 -435.109,E2 -435.109} C_VEL
LIN {X 0,Y 608.453,Z 346.617,A -85,B 0,C 180,E1 -436.963,E2 -436.963} C_VEL
LIN {X 0,Y 608.559,Z 408.003,A -85,B 0,C 180,E1 -437.707,E2 -437.707} C_VEL
LIN {X 0,Y 608.522,Z 454.975,A -85,B 0,C 180,E1 -438.277,E2 -438.277} C_VEL
LIN {X 0,Y 608.491,Z 468.235,A -85,B 0,C 180,E1 -438.572,E2 -438.572} C_VEL
LIN {X 0,Y 608.51,Z 480.659,A -85,B 0,C 180,E1 -438.983,E2 -438.983} C_VEL
LIN {X 0,Y 608.514,Z 492.644,A -85,B 0,C 180,E1 -439.52,E2 -439.52} C_VEL
LIN {X 0,Y 608.471,Z 504.205,A -85,B 0,C 180,E1 -440.191,E2 -440.191} C_VEL
LIN {X 0,Y 608.485,Z 514.6,A -85,B 0,C 180,E1 -440.946,E2 -440.946} C_VEL
LIN {X 0,Y 608.459,Z 523.007,A -85,B 0,C 180,E1 -441.699,E2 -441.699} C_VEL
LIN {X 0,Y 608.47,Z 530.964,A -85,B 0,C 180,E1 -442.534,E2 -442.534} C_VEL
LIN {X 0,Y 608.436,Z 538.301,A -85,B 0,C 180,E1 -443.486,E2 -443.486} C_VEL
LIN {X 0,Y 608.45,Z 543.868,A -85,B 0,C 180,E1 -444.366,E2 -444.366} C_VEL
LIN {X 0,Y 608.432,Z 548.952,A -85,B 0,C 180,E1 -445.363,E2 -445.363} C_VEL
LIN {X 0,Y 608.449,Z 552.897,A -85,B 0,C 180,E1 -446.358,E2 -446.358} C_VEL
LIN {X 0,Y 608.425,Z 555.81,A -85,B 0,C 180,E1 -447.352,E2 -447.352} C_VEL
LIN {X 0,Y 608.442,Z 557.202,A -85,B 0,C 180,E1 -448.015,E2 -448.015} C_VEL
LIN {X 0,Y 608.438,Z 558.784,A -85,B 0,C 180,E1 -449.339,E2 -449.339} C_VEL
LIN {X 0,Y 608.434,Z 559,A -85,B 0,C 180,E1 -450,E2 -450} C_VEL
LIN {X 0,Y 608.448,Z 558.183,A -85,B 0,C 180,E1 -451.324,E2 -451.324} C_VEL
LIN {X 0,Y 608.442,Z 557.201,A -85,B 0,C 180,E1 -451.986,E2 -451.986} C_VEL
LIN {X 0,Y 608.425,Z 555.808,A -85,B 0,C 180,E1 -452.649,E2 -452.649} C_VEL
LIN {X 0,Y 608.449,Z 552.895,A -85,B 0,C 180,E1 -453.643,E2 -453.643} C_VEL
LIN {X 0,Y 608.432,Z 548.949,A -85,B 0,C 180,E1 -454.638,E2 -454.638} C_VEL
LIN {X 0,Y 608.437,Z 542.875,A -85,B 0,C 180,E1 -455.801,E2 -455.801} C_VEL
LIN {X 0,Y 608.461,Z 536.233,A -85,B 0,C 180,E1 -456.8,E2 -456.8} C_VEL
LIN {X 0,Y 608.456,Z 527.987,A -85,B 0,C 180,E1 -457.8,E2 -457.8} C_VEL
LIN {X 0,Y 608.477,Z 517.596,A -85,B 0,C 180,E1 -458.803,E2 -458.803} C_VEL
LIN {X 0,Y 608.488,Z 506.744,A -85,B 0,C 180,E1 -459.641,E2 -459.641} C_VEL
LIN {X 0,Y 608.492,Z 495.769,A -85,B 0,C 180,E1 -460.313,E2 -460.313} C_VEL
LIN {X 0,Y 608.534,Z 483.808,A -85,B 0,C 180,E1 -460.888,E2 -460.888} C_VEL
LIN {X 0,Y 608.506,Z 471.873,A -85,B 0,C 180,E1 -461.323,E2 -461.323} C_VEL
LIN {X 0,Y 608.507,Z 459.501,A -85,B 0,C 180,E1 -461.64,E2 -461.64} C_VEL
LIN {X 0,Y 608.531,Z 443.716,A -85,B 0,C 180,E1 -461.872,E2 -461.872} C_VEL
LIN {X 0,Y 608.508,Z 347.127,A -85,B 0,C 180,E1 -463.016,E2 -463.016} C_VEL
LIN {X 0,Y 608.454,Z 346.126,A -85,B 0,C 180,E1 -463.102,E2 -463.102} C_VEL
LIN {X 0,Y 608.467,Z 327.357,A -85,B 0,C 180,E1 -465.578,E2 -465.578} C_VEL
LIN {X 0,Y 608.508,Z 307.94,A -85,B 0,C 180,E1 -468.17,E2 -468.17} C_VEL
LIN {X 0,Y 608.553,Z 287.229,A -85,B 0,C 180,E1 -470.978,E2 -470.978} C_VEL
LIN {X 0,Y 608.461,Z 274.687,A -85,B 0,C 180,E1 -472.715,E2 -472.715} C_VEL
LIN {X 0,Y 608.441,Z 274.689,A -85,B 0,C 180,E1 -475.301,E2 -475.301} C_VEL
LIN {X 0,Y 608.445,Z 274.69,A -85,B 0,C 180,E1 -477.518,E2 -477.518} C_VEL
LIN {X 0,Y 608.464,Z 274.694,A -85,B 0,C 180,E1 -479.971,E2 -479.971} C_VEL
LIN {X 0,Y 608.454,Z 274.687,A -85,B 0,C 180,E1 -482.88,E2 -482.88} C_VEL
LIN {X 0,Y 608.433,Z 274.689,A -85,B 0,C 180,E1 -485.278,E2 -485.278} C_VEL
LIN {X 0,Y 608.463,Z 274.687,A -85,B 0,C 180,E1 -487.747,E2 -487.747} C_VEL
LIN {X 0,Y 608.446,Z 274.697,A -85,B 0,C 180,E1 -490.328,E2 -490.328} C_VEL
LIN {X 0,Y 608.474,Z 274.684,A -85,B 0,C 180,E1 -493.309,E2 -493.309} C_VEL
LIN {X 0,Y 608.46,Z 274.688,A -85,B 0,C 180,E1 -496.129,E2 -496.129} C_VEL
LIN {X 0,Y 608.453,Z 274.696,A -85,B 0,C 180,E1 -498.823,E2 -498.823} C_VEL
LIN {X 0,Y 608.464,Z 274.685,A -85,B 0,C 180,E1 -501.76,E2 -501.76} C_VEL
LIN {X 0,Y 608.444,Z 274.687,A -85,B 0,C 180,E1 -503.954,E2 -503.954} C_VEL
LIN {X 0,Y 608.443,Z 274.689,A -85,B 0,C 180,E1 -506.328,E2 -506.328} C_VEL
LIN {X 0,Y 608.444,Z 274.693,A -85,B 0,C 180,E1 -508.732,E2 -508.732} C_VEL
LIN {X 0,Y 608.469,Z 274.691,A -85,B 0,C 180,E1 -511.38,E2 -511.38} C_VEL
LIN {X 0,Y 608.469,Z 274.684,A -85,B 0,C 180,E1 -514.279,E2 -514.279} C_VEL
LIN {X 0,Y 608.45,Z 274.691,A -85,B 0,C 180,E1 -516.876,E2 -516.876} C_VEL
LIN {X 0,Y 608.459,Z 274.691,A -85,B 0,C 180,E1 -519.726,E2 -519.726} C_VEL
LIN {X 0,Y 608.447,Z 274.691,A -85,B 0,C 180,E1 -521.828,E2 -521.828} C_VEL
LIN {X 0,Y 608.464,Z 274.685,A -85,B 0,C 180,E1 -524.594,E2 -524.594} C_VEL
LIN {X 0,Y 608.472,Z 274.69,A -85,B 0,C 180,E1 -527.323,E2 -527.323} C_VEL
LIN {X 0,Y 608.448,Z 274.692,A -85,B 0,C 180,E1 -530.022,E2 -530.022} C_VEL
LIN {X 0,Y 608.462,Z 274.685,A -85,B 0,C 180,E1 -532.7,E2 -532.7} C_VEL
LIN {X 0,Y 608.443,Z 274.69,A -85,B 0,C 180,E1 -535.362,E2 -535.362} C_VEL
LIN {X 0,Y 608.461,Z 274.696,A -85,B 0,C 180,E1 -538.014,E2 -538.014} C_VEL
LIN {X 0,Y 608.47,Z 274.686,A -85,B 0,C 180,E1 -540.662,E2 -540.662} C_VEL
LIN {X 0,Y 608.479,Z 274.683,A -85,B 0,C 180,E1 -543.311,E2 -543.311} C_VEL
LIN {X 0,Y 608.453,Z 274.693,A -85,B 0,C 180,E1 -545.967,E2 -545.967} C_VEL
LIN {X 0,Y 608.453,Z 274.691,A -85,B 0,C 180,E1 -548.636,E2 -548.636} C_VEL
LIN {X 0,Y 608.459,Z 274.686,A -85,B 0,C 180,E1 -549.453,E2 -549.453} C_VEL
LIN {X 0,Y 607.773,Z 274.778,A -85,B 0,C 180,E1 -550.005,E2 -550.005} C_VEL
LIN {X 0,Y 604.916,Z 275.134,A -85,B 0,C 180,E1 -550.902,E2 -550.902} C_VEL
LIN {X 0,Y 602.515,Z 275.433,A -85,B 0,C 180,E1 -551.624,E2 -551.624} C_VEL
LIN {X 0,Y 601.487,Z 275.561,A -85,B 0,C 180,E1 -552.18,E2 -552.18} C_VEL
LIN {X 0,Y 601.404,Z 275.569,A -85,B 0,C 180,E1 -552.369,E2 -552.369} C_VEL
LIN {X 0,Y 601.429,Z 275.565,A -85,B 0,C 180,E1 -554.897,E2 -554.897} C_VEL
LIN {X 0,Y 601.428,Z 275.565,A -85,B 0,C 180,E1 -556.986,E2 -556.986} C_VEL
LIN {X 0,Y 601.4,Z 275.565,A -85,B 0,C 180,E1 -559.81,E2 -559.81} C_VEL
LIN {X 0,Y 601.413,Z 275.573,A -85,B 0,C 180,E1 -562.606,E2 -562.606} C_VEL
LIN {X 0,Y 601.398,Z 275.575,A -85,B 0,C 180,E1 -564.879,E2 -564.879} C_VEL
LIN {X 0,Y 601.412,Z 275.566,A -85,B 0,C 180,E1 -567.362,E2 -567.362} C_VEL
LIN {X 0,Y 601.427,Z 275.562,A -85,B 0,C 180,E1 -570.164,E2 -570.164} C_VEL
LIN {X 0,Y 601.416,Z 275.568,A -85,B 0,C 180,E1 -572.715,E2 -572.715} C_VEL
LIN {X 0,Y 601.392,Z 275.578,A -85,B 0,C 180,E1 -575.112,E2 -575.112} C_VEL
LIN {X 0,Y 601.434,Z 275.568,A -85,B 0,C 180,E1 -577.419,E2 -577.419} C_VEL
LIN {X 0,Y 601.4,Z 275.566,A -85,B 0,C 180,E1 -579.996,E2 -579.996} C_VEL
LIN {X 0,Y 601.412,Z 275.565,A -85,B 0,C 180,E1 -582.67,E2 -582.67} C_VEL
LIN {X 0,Y 601.397,Z 275.577,A -85,B 0,C 180,E1 -585.48,E2 -585.48} C_VEL
LIN {X 0,Y 601.423,Z 275.562,A -85,B 0,C 180,E1 -588.407,E2 -588.407} C_VEL
LIN {X 0,Y 601.428,Z 275.571,A -85,B 0,C 180,E1 -591.53,E2 -591.53} C_VEL
LIN {X 0,Y 601.384,Z 275.57,A -85,B 0,C 180,E1 -594.245,E2 -594.245} C_VEL
LIN {X 0,Y 601.415,Z 275.564,A -85,B 0,C 180,E1 -596.686,E2 -596.686} C_VEL
LIN {X 0,Y 601.415,Z 275.564,A -85,B 0,C 180,E1 -599.058,E2 -599.058} C_VEL
LIN {X 0,Y 601.421,Z 275.577,A -85,B 0,C 180,E1 -601.242,E2 -601.242} C_VEL
LIN {X 0,Y 601.482,Z 289.401,A -85,B 0,C 180,E1 -603.64,E2 -603.64} C_VEL
LIN {X 0,Y 601.377,Z 305.585,A -85,B 0,C 180,E1 -606.405,E2 -606.405} C_VEL
LIN {X 0,Y 601.383,Z 308.404,A -85,B 0,C 180,E1 -606.884,E2 -606.884} C_VEL
LIN {X 0,Y 601.696,Z 314.283,A -85,B 0,C 180,E1 -606.965,E2 -606.965} C_VEL
LIN {X 0,Y 601.552,Z 414.84,A -85,B 0,C 180,E1 -608.181,E2 -608.181} C_VEL
LIN {X 0,Y 601.504,Z 427.885,A -85,B 0,C 180,E1 -608.472,E2 -608.472} C_VEL
LIN {X 0,Y 601.548,Z 440.536,A -85,B 0,C 180,E1 -608.894,E2 -608.894} C_VEL
LIN {X 0,Y 601.502,Z 451.857,A -85,B 0,C 180,E1 -609.401,E2 -609.401} C_VEL
LIN {X 0,Y 601.444,Z 462.594,A -85,B 0,C 180,E1 -610.014,E2 -610.014} C_VEL
LIN {X 0,Y 601.444,Z 473.712,A -85,B 0,C 180,E1 -610.813,E2 -610.813} C_VEL
LIN {X 0,Y 601.434,Z 482.641,A -85,B 0,C 180,E1 -611.609,E2 -611.609} C_VEL
LIN {X 0,Y 601.408,Z 490.933,A -85,B 0,C 180,E1 -612.487,E2 -612.487} C_VEL
LIN {X 0,Y 601.394,Z 498.448,A -85,B 0,C 180,E1 -613.477,E2 -613.477} C_VEL
LIN {X 0,Y 601.342,Z 504.206,A -85,B 0,C 180,E1 -614.407,E2 -614.407} C_VEL
LIN {X 0,Y 601.333,Z 509.349,A -85,B 0,C 180,E1 -615.447,E2 -615.447} C_VEL
LIN {X 0,Y 601.341,Z 513.286,A -85,B 0,C 180,E1 -616.482,E2 -616.482} C_VEL
LIN {X 0,Y 601.327,Z 515.295,A -85,B 0,C 180,E1 -617.17,E2 -617.17} C_VEL
LIN {X 0,Y 601.342,Z 516.872,A -85,B 0,C 180,E1 -617.856,E2 -617.856} C_VEL
LIN {X 0,Y 601.352,Z 518.538,A -85,B 0,C 180,E1 -619.025,E2 -619.025} C_VEL
LIN {X 0,Y 601.328,Z 518.973,A -85,B 0,C 180,E1 -619.903,E2 -619.903} C_VEL
LIN {X 0,Y 601.335,Z 518.872,A -85,B 0,C 180,E1 -620.583,E2 -620.583} C_VEL
LIN {X 0,Y 601.33,Z 517.393,A -85,B 0,C 180,E1 -621.938,E2 -621.938} C_VEL
LIN {X 0,Y 601.322,Z 516.062,A -85,B 0,C 180,E1 -622.613,E2 -622.613} C_VEL
LIN {X 0,Y 601.353,Z 513.908,A -85,B 0,C 180,E1 -623.41,E2 -623.41} C_VEL
LIN {X 0,Y 601.351,Z 509.384,A -85,B 0,C 180,E1 -624.635,E2 -624.635} C_VEL
LIN {X 0,Y 601.358,Z 504.422,A -85,B 0,C 180,E1 -625.643,E2 -625.643} C_VEL
LIN {X 0,Y 601.352,Z 498.208,A -85,B 0,C 180,E1 -626.65,E2 -626.65} C_VEL
LIN {X 0,Y 601.395,Z 490.471,A -85,B 0,C 180,E1 -627.656,E2 -627.656} C_VEL
LIN {X 0,Y 601.434,Z 480.841,A -85,B 0,C 180,E1 -628.66,E2 -628.66} C_VEL
LIN {X 0,Y 601.448,Z 470.908,A -85,B 0,C 180,E1 -629.498,E2 -629.498} C_VEL
LIN {X 0,Y 601.483,Z 459.729,A -85,B 0,C 180,E1 -630.251,E2 -630.251} C_VEL
LIN {X 0,Y 601.512,Z 448.824,A -85,B 0,C 180,E1 -630.836,E2 -630.836} C_VEL
LIN {X 0,Y 601.559,Z 436.76,A -85,B 0,C 180,E1 -631.339,E2 -631.339} C_VEL
LIN {X 0,Y 601.544,Z 424.152,A -85,B 0,C 180,E1 -631.715,E2 -631.715} C_VEL
LIN {X 0,Y 601.577,Z 410.887,A -85,B 0,C 180,E1 -631.966,E2 -631.966} C_VEL
LIN {X 0,Y 601.487,Z 309.302,A -85,B 0,C 180,E1 -633.189,E2 -633.189} C_VEL
LIN {X 0,Y 601.384,Z 308.298,A -85,B 0,C 180,E1 -633.224,E2 -633.224} C_VEL
LIN {X 0,Y 601.383,Z 295.741,A -85,B 0,C 180,E1 -635.364,E2 -635.364} C_VEL
LIN {X 0,Y 601.431,Z 282.044,A -85,B 0,C 180,E1 -637.722,E2 -637.722} C_VEL
LIN {X 0,Y 601.37,Z 275.572,A -85,B 0,C 180,E1 -638.865,E2 -638.865} C_VEL
LIN {X 0,Y 601.368,Z 275.57,A -85,B 0,C 180,E1 -641.459,E2 -641.459} C_VEL
LIN {X 0,Y 601.401,Z 275.575,A -85,B 0,C 180,E1 -644.205,E2 -644.205} C_VEL
LIN {X 0,Y 601.397,Z 275.567,A -85,B 0,C 180,E1 -646.986,E2 -646.986} C_VEL
LIN {X 0,Y 601.371,Z 275.57,A -85,B 0,C 180,E1 -649.81,E2 -649.81} C_VEL
LIN {X 0,Y 601.379,Z 275.57,A -85,B 0,C 180,E1 -651.96,E2 -651.96} C_VEL
LIN {X 0,Y 601.38,Z 275.573,A -85,B 0,C 180,E1 -654.879,E2 -654.879} C_VEL
LIN {X 0,Y 601.382,Z 275.568,A -85,B 0,C 180,E1 -657.356,E2 -657.356} C_VEL
LIN {X 0,Y 601.374,Z 275.569,A -85,B 0,C 180,E1 -659.395,E2 -659.395} C_VEL
LIN {X 0,Y 601.379,Z 275.568,A -85,B 0,C 180,E1 -661.727,E2 -661.727} C_VEL
LIN {X 0,Y 601.402,Z 275.566,A -85,B 0,C 180,E1 -664.119,E2 -664.119} C_VEL
LIN {X 0,Y 601.43,Z 275.564,A -85,B 0,C 180,E1 -667.381,E2 -667.381} C_VEL
LIN {X 0,Y 601.372,Z 275.568,A -85,B 0,C 180,E1 -669.997,E2 -669.997} C_VEL
LIN {X 0,Y 601.374,Z 275.573,A -85,B 0,C 180,E1 -672.672,E2 -672.672} C_VEL
LIN {X 0,Y 601.419,Z 275.568,A -85,B 0,C 180,E1 -675.464,E2 -675.464} C_VEL
LIN {X 0,Y 601.399,Z 275.565,A -85,B 0,C 180,E1 -678.408,E2 -678.408} C_VEL
LIN {X 0,Y 601.423,Z 275.569,A -85,B 0,C 180,E1 -681.529,E2 -681.529} C_VEL
LIN {X 0,Y 601.372,Z 275.569,A -85,B 0,C 180,E1 -684.244,E2 -684.244} C_VEL
LIN {X 0,Y 601.403,Z 275.565,A -85,B 0,C 180,E1 -686.685,E2 -686.685} C_VEL
LIN {X 0,Y 601.399,Z 275.569,A -85,B 0,C 180,E1 -689.057,E2 -689.057} C_VEL
LIN {X 0,Y 601.424,Z 275.57,A -85,B 0,C 180,E1 -691.373,E2 -691.373} C_VEL
LIN {X 0,Y 601.403,Z 275.565,A -85,B 0,C 180,E1 -694.381,E2 -694.381} C_VEL
LIN {X 0,Y 601.385,Z 275.567,A -85,B 0,C 180,E1 -696.588,E2 -696.588} C_VEL
LIN {X 0,Y 601.416,Z 275.569,A -85,B 0,C 180,E1 -699.478,E2 -699.478} C_VEL
LIN {X 0,Y 601.386,Z 275.57,A -85,B 0,C 180,E1 -702.311,E2 -702.311} C_VEL
LIN {X 0,Y 601.411,Z 275.566,A -85,B 0,C 180,E1 -704.409,E2 -704.409} C_VEL
LIN {X 0,Y 601.398,Z 275.566,A -85,B 0,C 180,E1 -707.171,E2 -707.171} C_VEL
LIN {X 0,Y 601.427,Z 275.57,A -85,B 0,C 180,E1 -709.905,E2 -709.905} C_VEL
LIN {X 0,Y 601.447,Z 275.562,A -85,B 0,C 180,E1 -712.615,E2 -712.615} C_VEL
LIN {X 0,Y 601.399,Z 275.565,A -85,B 0,C 180,E1 -715.308,E2 -715.308} C_VEL
LIN {X 0,Y 601.414,Z 275.57,A -85,B 0,C 180,E1 -717.991,E2 -717.991} C_VEL
LIN {X 0,Y 601.45,Z 275.564,A -85,B 0,C 180,E1 -720.67,E2 -720.67} C_VEL
LIN {X 0,Y 601.424,Z 275.562,A -85,B 0,C 180,E1 -723.35,E2 -723.35} C_VEL
LIN {X 0,Y 601.393,Z 275.57,A -85,B 0,C 180,E1 -726.037,E2 -726.037} C_VEL
LIN {X 0,Y 601.437,Z 275.568,A -85,B 0,C 180,E1 -728.738,E2 -728.738} C_VEL
LIN {X 0,Y 601.428,Z 275.562,A -85,B 0,C 180,E1 -731.458,E2 -731.458} C_VEL
LIN {X 0,Y 601.41,Z 275.567,A -85,B 0,C 180,E1 -734.206,E2 -734.206} C_VEL
LIN {X 0,Y 601.426,Z 275.569,A -85,B 0,C 180,E1 -736.986,E2 -736.986} C_VEL
LIN {X 0,Y 601.397,Z 275.565,A -85,B 0,C 180,E1 -739.81,E2 -739.81} C_VEL
LIN {X 0,Y 601.405,Z 275.571,A -85,B 0,C 180,E1 -742.683,E2 -742.683} C_VEL
LIN {X 0,Y 601.398,Z 275.575,A -85,B 0,C 180,E1 -744.879,E2 -744.879} C_VEL
LIN {X 0,Y 601.414,Z 275.564,A -85,B 0,C 180,E1 -747.868,E2 -747.868} C_VEL
LIN {X 0,Y 601.442,Z 275.56,A -85,B 0,C 180,E1 -750.163,E2 -750.163} C_VEL
LIN {X 0,Y 601.413,Z 275.567,A -85,B 0,C 180,E1 -752.716,E2 -752.716} C_VEL
LIN {X 0,Y 601.389,Z 275.575,A -85,B 0,C 180,E1 -755.113,E2 -755.113} C_VEL
LIN {X 0,Y 601.43,Z 275.571,A -85,B 0,C 180,E1 -757.42,E2 -757.42} C_VEL
LIN {X 0,Y 601.404,Z 275.566,A -85,B 0,C 180,E1 -759.996,E2 -759.996} C_VEL
LIN {X 0,Y 601.409,Z 275.564,A -85,B 0,C 180,E1 -762.671,E2 -762.671} C_VEL
LIN {X 0,Y 601.422,Z 275.573,A -85,B 0,C 180,E1 -765.483,E2 -765.483} C_VEL
LIN {X 0,Y 601.423,Z 275.563,A -85,B 0,C 180,E1 -768.407,E2 -768.407} C_VEL
LIN {X 0,Y 601.428,Z 275.57,A -85,B 0,C 180,E1 -771.53,E2 -771.53} C_VEL
LIN {X 0,Y 601.383,Z 275.57,A -85,B 0,C 180,E1 -774.246,E2 -774.246} C_VEL
LIN {X 0,Y 601.415,Z 275.563,A -85,B 0,C 180,E1 -776.687,E2 -776.687} C_VEL
LIN {X 0,Y 601.414,Z 275.563,A -85,B 0,C 180,E1 -779.059,E2 -779.059} C_VEL
LIN {X 0,Y 601.429,Z 275.564,A -85,B 0,C 180,E1 -781.374,E2 -781.374} C_VEL
LIN {X 0,Y 601.399,Z 275.57,A -85,B 0,C 180,E1 -783.637,E2 -783.637} C_VEL
LIN {X 0,Y 601.418,Z 275.57,A -85,B 0,C 180,E1 -786.59,E2 -786.59} C_VEL
LIN {X 0,Y 601.422,Z 275.584,A -85,B 0,C 180,E1 -787.137,E2 -787.137} C_VEL
LIN {X 0,Y 601.697,Z 280.78,A -85,B 0,C 180,E1 -787.875,E2 -787.875} C_VEL
LIN {X 0,Y 601.601,Z 302.767,A -85,B 0,C 180,E1 -790.908,E2 -790.908} C_VEL
LIN {X 0,Y 601.524,Z 323.479,A -85,B 0,C 180,E1 -793.716,E2 -793.716} C_VEL
LIN {X 0,Y 601.468,Z 344.19,A -85,B 0,C 180,E1 -796.486,E2 -796.486} C_VEL
LIN {X 0,Y 601.426,Z 346.617,A -85,B 0,C 180,E1 -796.807,E2 -796.807} C_VEL
LIN {X 0,Y 601.665,Z 352.554,A -85,B 0,C 180,E1 -796.899,E2 -796.899} C_VEL
LIN {X 0,Y 601.594,Z 454.975,A -85,B 0,C 180,E1 -798.14,E2 -798.14} C_VEL
LIN {X 0,Y 601.556,Z 468.236,A -85,B 0,C 180,E1 -798.438,E2 -798.438} C_VEL
LIN {X 0,Y 601.539,Z 480.658,A -85,B 0,C 180,E1 -798.854,E2 -798.854} C_VEL
LIN {X 0,Y 601.521,Z 492.643,A -85,B 0,C 180,E1 -799.397,E2 -799.397} C_VEL
LIN {X 0,Y 601.472,Z 504.206,A -85,B 0,C 180,E1 -800.076,E2 -800.076} C_VEL
LIN {X 0,Y 601.444,Z 514.601,A -85,B 0,C 180,E1 -800.839,E2 -800.839} C_VEL
LIN {X 0,Y 601.404,Z 523.02,A -85,B 0,C 180,E1 -801.601,E2 -801.601} C_VEL
LIN {X 0,Y 601.417,Z 530.964,A -85,B 0,C 180,E1 -802.446,E2 -802.446} C_VEL
LIN {X 0,Y 601.365,Z 538.251,A -85,B 0,C 180,E1 -803.402,E2 -803.402} C_VEL
LIN {X 0,Y 601.371,Z 543.868,A -85,B 0,C 180,E1 -804.299,E2 -804.299} C_VEL
LIN {X 0,Y 601.336,Z 548.952,A -85,B 0,C 180,E1 -805.308,E2 -805.308} C_VEL
LIN {X 0,Y 601.367,Z 552.897,A -85,B 0,C 180,E1 -806.315,E2 -806.315} C_VEL
LIN {X 0,Y 601.325,Z 555.81,A -85,B 0,C 180,E1 -807.321,E2 -807.321} C_VEL
LIN {X 0,Y 601.341,Z 557.202,A -85,B 0,C 180,E1 -807.991,E2 -807.991} C_VEL
LIN {X 0,Y 601.339,Z 558.784,A -85,B 0,C 180,E1 -809.331,E2 -809.331} C_VEL
LIN {X 0,Y 601.335,Z 559,A -85,B 0,C 180,E1 -810,E2 -810} C_VEL
LIN {X 0,Y 601.347,Z 558.184,A -85,B 0,C 180,E1 -811.34,E2 -811.34} C_VEL
LIN {X 0,Y 601.341,Z 557.201,A -85,B 0,C 180,E1 -812.01,E2 -812.01} C_VEL
LIN {X 0,Y 601.325,Z 555.809,A -85,B 0,C 180,E1 -812.68,E2 -812.68} C_VEL
LIN {X 0,Y 601.367,Z 552.895,A -85,B 0,C 180,E1 -813.686,E2 -813.686} C_VEL
LIN {X 0,Y 601.336,Z 548.949,A -85,B 0,C 180,E1 -814.693,E2 -814.693} C_VEL
LIN {X 0,Y 601.372,Z 542.875,A -85,B 0,C 180,E1 -815.869,E2 -815.869} C_VEL
LIN {X 0,Y 601.381,Z 536.234,A -85,B 0,C 180,E1 -816.88,E2 -816.88} C_VEL
LIN {X 0,Y 601.4,Z 527.987,A -85,B 0,C 180,E1 -817.893,E2 -817.893} C_VEL
LIN {X 0,Y 601.435,Z 517.596,A -85,B 0,C 180,E1 -818.907,E2 -818.907} C_VEL
LIN {X 0,Y 601.46,Z 506.744,A -85,B 0,C 180,E1 -819.755,E2 -819.755} C_VEL
LIN {X 0,Y 601.494,Z 495.771,A -85,B 0,C 180,E1 -820.434,E2 -820.434} C_VEL
LIN {X 0,Y 601.549,Z 483.679,A -85,B 0,C 180,E1 -821.022,E2 -821.022} C_VEL
LIN {X 0,Y 601.53,Z 471.871,A -85,B 0,C 180,E1 -821.456,E2 -821.456} C_VEL
LIN {X 0,Y 601.577,Z 459.5,A -85,B 0,C 180,E1 -821.776,E2 -821.776} C_VEL
LIN {X 0,Y 601.608,Z 443.716,A -85,B 0,C 180,E1 -822.01,E2 -822.01} C_VEL
LIN {X 0,Y 601.479,Z 347.127,A -85,B 0,C 180,E1 -823.171,E2 -823.171} C_VEL
LIN {X 0,Y 601.461,Z 346.126,A -85,B 0,C 180,E1 -823.257,E2 -823.257} C_VEL
LIN {X 0,Y 601.467,Z 326.062,A -85,B 0,C 180,E1 -825.938,E2 -825.938} C_VEL
LIN {X 0,Y 601.574,Z 306.208,A -85,B 0,C 180,E1 -828.623,E2 -828.623} C_VEL
LIN {X 0,Y 601.654,Z 284.64,A -85,B 0,C 180,E1 -831.59,E2 -831.59} C_VEL
LIN {X 0,Y 601.629,Z 276.873,A -85,B 0,C 180,E1 -832.674,E2 -832.674} C_VEL
LIN {X 0,Y 601.417,Z 275.567,A -85,B 0,C 180,E1 -832.887,E2 -832.887} C_VEL
LIN {X 0,Y 601.398,Z 275.566,A -85,B 0,C 180,E1 -834.879,E2 -834.879} C_VEL
LIN {X 0,Y 601.412,Z 275.565,A -85,B 0,C 180,E1 -837.361,E2 -837.361} C_VEL
LIN {X 0,Y 601.431,Z 275.573,A -85,B 0,C 180,E1 -840.164,E2 -840.164} C_VEL
LIN {X 0,Y 601.421,Z 275.565,A -85,B 0,C 180,E1 -842.715,E2 -842.715} C_VEL
LIN {X 0,Y 601.391,Z 275.566,A -85,B 0,C 180,E1 -845.111,E2 -845.111} C_VEL
LIN {X 0,Y 601.435,Z 275.561,A -85,B 0,C 180,E1 -847.419,E2 -847.419} C_VEL
LIN {X 0,Y 601.401,Z 275.569,A -85,B 0,C 180,E1 -849.996,E2 -849.996} C_VEL
LIN {X 0,Y 601.41,Z 275.573,A -85,B 0,C 180,E1 -852.67,E2 -852.67} C_VEL
LIN {X 0,Y 601.398,Z 275.565,A -85,B 0,C 180,E1 -855.479,E2 -855.479} C_VEL
LIN {X 0,Y 601.422,Z 275.568,A -85,B 0,C 180,E1 -858.407,E2 -858.407} C_VEL
LIN {X 0,Y 601.431,Z 275.562,A -85,B 0,C 180,E1 -861.529,E2 -861.529} C_VEL
LIN {X 0,Y 601.383,Z 275.568,A -85,B 0,C 180,E1 -864.245,E2 -864.245} C_VEL
LIN {X 0,Y 601.413,Z 275.569,A -85,B 0,C 180,E1 -866.685,E2 -866.685} C_VEL
LIN {X 0,Y 601.414,Z 275.575,A -85,B 0,C 180,E1 -869.057,E2 -869.057} C_VEL
LIN {X 0,Y 601.429,Z 275.568,A -85,B 0,C 180,E1 -871.373,E2 -871.373} C_VEL
LIN {X 0,Y 601.41,Z 275.564,A -85,B 0,C 180,E1 -874.132,E2 -874.132} C_VEL
LIN {X 0,Y 601.418,Z 275.564,A -85,B 0,C 180,E1 -876.589,E2 -876.589} C_VEL
LIN {X 0,Y 601.429,Z 275.571,A -85,B 0,C 180,E1 -879.478,E2 -879.478} C_VEL
LIN {X 0,Y 601.39,Z 275.566,A -85,B 0,C 180,E1 -882.311,E2 -882.311} C_VEL
LIN {X 0,Y 601.408,Z 275.564,A -85,B 0,C 180,E1 -884.408,E2 -884.408} C_VEL
LIN {X 0,Y 601.416,Z 275.566,A -85,B 0,C 180,E1 -887.172,E2 -887.172} C_VEL
LIN {X 0,Y 601.427,Z 275.569,A -85,B 0,C 180,E1 -889.905,E2 -889.905} C_VEL
LIN {X 0,Y 601.439,Z 275.56,A -85,B 0,C 180,E1 -892.615,E2 -892.615} C_VEL
LIN {X 0,Y 601.413,Z 275.565,A -85,B 0,C 180,E1 -895.308,E2 -895.308} C_VEL
LIN {X 0,Y 601.43,Z 275.572,A -85,B 0,C 180,E1 -897.991,E2 -897.991} C_VEL
LIN {X 0,Y 601.442,Z 275.561,A -85,B 0,C 180,E1 -900.669,E2 -900.669} C_VEL
LIN {X 0,Y 601.43,Z 275.561,A -85,B 0,C 180,E1 -903.349,E2 -903.349} C_VEL
LIN {X 0,Y 601.405,Z 275.573,A -85,B 0,C 180,E1 -906.037,E2 -906.037} C_VEL
LIN {X 0,Y 601.414,Z 275.567,A -85,B 0,C 180,E1 -908.738,E2 -908.738} C_VEL
LIN {X 0,Y 601.431,Z 275.561,A -85,B 0,C 180,E1 -911.458,E2 -911.458} C_VEL
LIN {X 0,Y 601.404,Z 275.569,A -85,B 0,C 180,E1 -912.369,E2 -912.369} C_VEL
LIN {X 0,Y 600.741,Z 275.651,A -85,B 0,C 180,E1 -912.928,E2 -912.928} C_VEL
LIN {X 0,Y 597.894,Z 276.004,A -85,B 0,C 180,E1 -913.836,E2 -913.836} C_VEL
LIN {X 0,Y 595.484,Z 276.312,A -85,B 0,C 180,E1 -914.566,E2 -914.566} C_VEL
LIN {X 0,Y 594.445,Z 276.433,A -85,B 0,C 180,E1 -915.13,E2 -915.13} C_VEL
LIN {X 0,Y 594.358,Z 276.442,A -85,B 0,C 180,E1 -915.321,E2 -915.321} C_VEL
LIN {X 0,Y 594.385,Z 276.44,A -85,B 0,C 180,E1 -917.193,E2 -917.193} C_VEL
LIN {X 0,Y 594.371,Z 276.442,A -85,B 0,C 180,E1 -920.054,E2 -920.054} C_VEL
LIN {X 0,Y 594.363,Z 276.448,A -85,B 0,C 180,E1 -922.967,E2 -922.967} C_VEL
LIN {X 0,Y 594.372,Z 276.445,A -85,B 0,C 180,E1 -925.193,E2 -925.193} C_VEL
LIN {X 0,Y 594.384,Z 276.44,A -85,B 0,C 180,E1 -927.527,E2 -927.527} C_VEL
LIN {X 0,Y 594.384,Z 276.44,A -85,B 0,C 180,E1 -930.328,E2 -930.328} C_VEL
LIN {X 0,Y 594.374,Z 276.449,A -85,B 0,C 180,E1 -932.95,E2 -932.95} C_VEL
LIN {X 0,Y 594.347,Z 276.45,A -85,B 0,C 180,E1 -935.409,E2 -935.409} C_VEL
LIN {X 0,Y 594.385,Z 276.44,A -85,B 0,C 180,E1 -937.941,E2 -937.941} C_VEL
LIN {X 0,Y 594.376,Z 276.443,A -85,B 0,C 180,E1 -940.822,E2 -940.822} C_VEL
LIN {X 0,Y 594.366,Z 276.451,A -85,B 0,C 180,E1 -943.3,E2 -943.3} C_VEL
LIN {X 0,Y 594.359,Z 276.443,A -85,B 0,C 180,E1 -946.161,E2 -946.161} C_VEL
LIN {X 0,Y 594.38,Z 276.439,A -85,B 0,C 180,E1 -948.536,E2 -948.536} C_VEL
LIN {X 0,Y 594.38,Z 276.445,A -85,B 0,C 180,E1 -951.296,E2 -951.296} C_VEL
LIN {X 0,Y 594.351,Z 276.454,A -85,B 0,C 180,E1 -953.756,E2 -953.756} C_VEL
LIN {X 0,Y 594.364,Z 276.445,A -85,B 0,C 180,E1 -956.238,E2 -956.238} C_VEL
LIN {X 0,Y 594.369,Z 276.442,A -85,B 0,C 180,E1 -958.65,E2 -958.65} C_VEL
LIN {X 0,Y 594.379,Z 276.46,A -85,B 0,C 180,E1 -961.167,E2 -961.167} C_VEL
LIN {X 0,Y 594.451,Z 289.692,A -85,B 0,C 180,E1 -963.491,E2 -963.491} C_VEL
LIN {X 0,Y 594.371,Z 304.836,A -85,B 0,C 180,E1 -966.112,E2 -966.112} C_VEL
LIN {X 0,Y 594.36,Z 308.38,A -85,B 0,C 180,E1 -966.722,E2 -966.722} C_VEL
LIN {X 0,Y 594.788,Z 313.177,A -85,B 0,C 180,E1 -966.797,E2 -966.797} C_VEL
LIN {X 0,Y 594.612,Z 415.343,A -85,B 0,C 180,E1 -968.05,E2 -968.05} C_VEL
LIN {X 0,Y 594.541,Z 428.208,A -85,B 0,C 180,E1 -968.344,E2 -968.344} C_VEL
LIN {X 0,Y 594.587,Z 441.107,A -85,B 0,C 180,E1 -968.784,E2 -968.784} C_VEL
LIN {X 0,Y 594.509,Z 452.709,A -85,B 0,C 180,E1 -969.319,E2 -969.319} C_VEL
LIN {X 0,Y 594.438,Z 463.403,A -85,B 0,C 180,E1 -969.948,E2 -969.948} C_VEL
LIN {X 0,Y 594.412,Z 474.795,A -85,B 0,C 180,E1 -970.791,E2 -970.791} C_VEL
LIN {X 0,Y 594.388,Z 483.185,A -85,B 0,C 180,E1 -971.561,E2 -971.561} C_VEL
LIN {X 0,Y 594.333,Z 491.368,A -85,B 0,C 180,E1 -972.45,E2 -972.45} C_VEL
LIN {X 0,Y 594.324,Z 499.198,A -85,B 0,C 180,E1 -973.512,E2 -973.512} C_VEL
LIN {X 0,Y 594.266,Z 505.424,A -85,B 0,C 180,E1 -974.568,E2 -974.568} C_VEL
LIN {X 0,Y 594.257,Z 510.301,A -85,B 0,C 180,E1 -975.62,E2 -975.62} C_VEL
LIN {X 0,Y 594.264,Z 513.993,A -85,B 0,C 180,E1 -976.667,E2 -976.667} C_VEL
LIN {X 0,Y 594.24,Z 516.616,A -85,B 0,C 180,E1 -977.708,E2 -977.708} C_VEL
LIN {X 0,Y 594.263,Z 518.519,A -85,B 0,C 180,E1 -978.989,E2 -978.989} C_VEL
LIN {X 0,Y 594.231,Z 518.946,A -85,B 0,C 180,E1 -979.781,E2 -979.781} C_VEL
LIN {X 0,Y 594.254,Z 518.909,A -85,B 0,C 180,E1 -980.469,E2 -980.469} C_VEL
LIN {X 0,Y 594.227,Z 518.466,A -85,B 0,C 180,E1 -981.155,E2 -981.155} C_VEL
LIN {X 0,Y 594.247,Z 516.314,A -85,B 0,C 180,E1 -982.525,E2 -982.525} C_VEL
LIN {X 0,Y 594.268,Z 514.006,A -85,B 0,C 180,E1 -983.419,E2 -983.419} C_VEL
LIN {X 0,Y 594.269,Z 509.882,A -85,B 0,C 180,E1 -984.571,E2 -984.571} C_VEL
LIN {X 0,Y 594.278,Z 505.056,A -85,B 0,C 180,E1 -985.591,E2 -985.591} C_VEL
LIN {X 0,Y 594.273,Z 498.99,A -85,B 0,C 180,E1 -986.61,E2 -986.61} C_VEL
LIN {X 0,Y 594.333,Z 491.468,A -85,B 0,C 180,E1 -987.628,E2 -987.628} C_VEL
LIN {X 0,Y 594.361,Z 483.721,A -85,B 0,C 180,E1 -988.475,E2 -988.475} C_VEL
LIN {X 0,Y 594.426,Z 474.51,A -85,B 0,C 180,E1 -989.322,E2 -989.322} C_VEL
LIN {X 0,Y 594.444,Z 464.254,A -85,B 0,C 180,E1 -990.084,E2 -990.084} C_VEL
LIN {X 0,Y 594.53,Z 452.879,A -85,B 0,C 180,E1 -990.762,E2 -990.762} C_VEL
LIN {X 0,Y 594.6,Z 440.947,A -85,B 0,C 180,E1 -991.312,E2 -991.312} C_VEL
LIN {X 0,Y 594.577,Z 427.819,A -85,B 0,C 180,E1 -991.756,E2 -991.756} C_VEL
LIN {X 0,Y 594.645,Z 414.604,A -85,B 0,C 180,E1 -992.053,E2 -992.053} C_VEL
LIN {X 0,Y 594.698,Z 310.83,A -85,B 0,C 180,E1 -993.324,E2 -993.324} C_VEL
LIN {X 0,Y 594.328,Z 308.386,A -85,B 0,C 180,E1 -993.368,E2 -993.368} C_VEL
LIN {X 0,Y 594.356,Z 296.445,A -85,B 0,C 180,E1 -995.428,E2 -995.428} C_VEL
LIN {X 0,Y 594.442,Z 282.747,A -85,B 0,C 180,E1 -997.814,E2 -997.814} C_VEL
LIN {X 0,Y 594.328,Z 276.45,A -85,B 0,C 180,E1 -998.928,E2 -998.928} C_VEL
LIN {X 0,Y 594.349,Z 276.446,A -85,B 0,C 180,E1 -1001.596,E2 -1001.596} C_VEL
LIN {X 0,Y 594.378,Z 276.45,A -85,B 0,C 180,E1 -1004.377,E2 -1004.377} C_VEL
LIN {X 0,Y 594.333,Z 276.446,A -85,B 0,C 180,E1 -1007.194,E2 -1007.194} C_VEL
LIN {X 0,Y 594.348,Z 276.444,A -85,B 0,C 180,E1 -1009.334,E2 -1009.334} C_VEL
LIN {X 0,Y 594.342,Z 276.444,A -85,B 0,C 180,E1 -1011.504,E2 -1011.504} C_VEL
LIN {X 0,Y 594.363,Z 276.451,A -85,B 0,C 180,E1 -1014.446,E2 -1014.446} C_VEL
LIN {X 0,Y 594.339,Z 276.445,A -85,B 0,C 180,E1 -1017.518,E2 -1017.518} C_VEL
LIN {X 0,Y 594.329,Z 276.446,A -85,B 0,C 180,E1 -1019.778,E2 -1019.778} C_VEL
LIN {X 0,Y 594.346,Z 276.445,A -85,B 0,C 180,E1 -1022.147,E2 -1022.147} C_VEL
LIN {X 0,Y 594.372,Z 276.447,A -85,B 0,C 180,E1 -1024.58,E2 -1024.58} C_VEL
LIN {X 0,Y 594.378,Z 276.441,A -85,B 0,C 180,E1 -1027.607,E2 -1027.607} C_VEL
LIN {X 0,Y 594.356,Z 276.446,A -85,B 0,C 180,E1 -1030.567,E2 -1030.567} C_VEL
LIN {X 0,Y 594.353,Z 276.45,A -85,B 0,C 180,E1 -1033.299,E2 -1033.299} C_VEL
LIN {X 0,Y 594.335,Z 276.445,A -85,B 0,C 180,E1 -1036.163,E2 -1036.163} C_VEL
LIN {X 0,Y 594.359,Z 276.443,A -85,B 0,C 180,E1 -1038.534,E2 -1038.534} C_VEL
LIN {X 0,Y 594.371,Z 276.452,A -85,B 0,C 180,E1 -1041.296,E2 -1041.296} C_VEL
LIN {X 0,Y 594.343,Z 276.448,A -85,B 0,C 180,E1 -1043.755,E2 -1043.755} C_VEL
LIN {X 0,Y 594.356,Z 276.443,A -85,B 0,C 180,E1 -1046.237,E2 -1046.237} C_VEL
LIN {X 0,Y 594.355,Z 276.443,A -85,B 0,C 180,E1 -1048.649,E2 -1048.649} C_VEL
LIN {X 0,Y 594.37,Z 276.444,A -85,B 0,C 180,E1 -1051.042,E2 -1051.042} C_VEL
LIN {X 0,Y 594.368,Z 276.445,A -85,B 0,C 180,E1 -1054.056,E2 -1054.056} C_VEL
LIN {X 0,Y 594.371,Z 276.442,A -85,B 0,C 180,E1 -1056.295,E2 -1056.295} C_VEL
LIN {X 0,Y 594.385,Z 276.441,A -85,B 0,C 180,E1 -1059.224,E2 -1059.224} C_VEL
LIN {X 0,Y 594.367,Z 276.448,A -85,B 0,C 180,E1 -1062.095,E2 -1062.095} C_VEL
LIN {X 0,Y 594.366,Z 276.447,A -85,B 0,C 180,E1 -1064.219,E2 -1064.219} C_VEL
LIN {X 0,Y 594.348,Z 276.443,A -85,B 0,C 180,E1 -1067.017,E2 -1067.017} C_VEL
LIN {X 0,Y 594.383,Z 276.446,A -85,B 0,C 180,E1 -1069.784,E2 -1069.784} C_VEL
LIN {X 0,Y 594.395,Z 276.442,A -85,B 0,C 180,E1 -1072.527,E2 -1072.527} C_VEL
LIN {X 0,Y 594.372,Z 276.44,A -85,B 0,C 180,E1 -1075.252,E2 -1075.252} C_VEL
LIN {X 0,Y 594.384,Z 276.445,A -85,B 0,C 180,E1 -1077.967,E2 -1077.967} C_VEL
LIN {X 0,Y 594.42,Z 276.44,A -85,B 0,C 180,E1 -1080.678,E2 -1080.678} C_VEL
LIN {X 0,Y 594.374,Z 276.44,A -85,B 0,C 180,E1 -1083.389,E2 -1083.389} C_VEL
LIN {X 0,Y 594.386,Z 276.439,A -85,B 0,C 180,E1 -1085.428,E2 -1085.428} C_VEL
LIN {X 0,Y 594.404,Z 276.441,A -85,B 0,C 180,E1 -1088.157,E2 -1088.157} C_VEL
LIN {X 0,Y 594.387,Z 276.442,A -85,B 0,C 180,E1 -1091.078,E2 -1091.078} C_VEL
LIN {X 0,Y 594.372,Z 276.44,A -85,B 0,C 180,E1 -1093.679,E2 -1093.679} C_VEL
LIN {X 0,Y 594.385,Z 276.45,A -85,B 0,C 180,E1 -1096.72,E2 -1096.72} C_VEL
LIN {X 0,Y 594.361,Z 276.445,A -85,B 0,C 180,E1 -1099.335,E2 -1099.335} C_VEL
LIN {X 0,Y 594.357,Z 276.444,A -85,B 0,C 180,E1 -1101.504,E2 -1101.504} C_VEL
LIN {X 0,Y 594.381,Z 276.442,A -85,B 0,C 180,E1 -1104.447,E2 -1104.447} C_VEL
LIN {X 0,Y 594.382,Z 276.444,A -85,B 0,C 180,E1 -1106.7,E2 -1106.7} C_VEL
LIN {X 0,Y 594.373,Z 276.45,A -85,B 0,C 180,E1 -1108.999,E2 -1108.999} C_VEL
LIN {X 0,Y 594.386,Z 276.442,A -85,B 0,C 180,E1 -1111.646,E2 -1111.646} C_VEL
LIN {X 0,Y 594.373,Z 276.442,A -85,B 0,C 180,E1 -1114.581,E2 -1114.581} C_VEL
LIN {X 0,Y 594.38,Z 276.447,A -85,B 0,C 180,E1 -1117.087,E2 -1117.087} C_VEL
LIN {X 0,Y 594.368,Z 276.445,A -85,B 0,C 180,E1 -1119.775,E2 -1119.775} C_VEL
LIN {X 0,Y 594.367,Z 276.441,A -85,B 0,C 180,E1 -1122.376,E2 -1122.376} C_VEL
LIN {X 0,Y 594.359,Z 276.447,A -85,B 0,C 180,E1 -1125.192,E2 -1125.192} C_VEL
LIN {X 0,Y 594.38,Z 276.442,A -85,B 0,C 180,E1 -1128.152,E2 -1128.152} C_VEL
LIN {X 0,Y 594.375,Z 276.443,A -85,B 0,C 180,E1 -1131.195,E2 -1131.195} C_VEL
LIN {X 0,Y 594.35,Z 276.455,A -85,B 0,C 180,E1 -1133.756,E2 -1133.756} C_VEL
LIN {X 0,Y 594.374,Z 276.444,A -85,B 0,C 180,E1 -1136.239,E2 -1136.239} C_VEL
LIN {X 0,Y 594.368,Z 276.442,A -85,B 0,C 180,E1 -1138.651,E2 -1138.651} C_VEL
LIN {X 0,Y 594.381,Z 276.44,A -85,B 0,C 180,E1 -1141.043,E2 -1141.043} C_VEL
LIN {X 0,Y 594.381,Z 276.451,A -85,B 0,C 180,E1 -1143.979,E2 -1143.979} C_VEL
LIN {X 0,Y 594.385,Z 276.446,A -85,B 0,C 180,E1 -1146.666,E2 -1146.666} C_VEL
LIN {X 0,Y 594.402,Z 276.555,A -85,B 0,C 180,E1 -1146.989,E2 -1146.989} C_VEL
LIN {X 0,Y 594.779,Z 282.056,A -85,B 0,C 180,E1 -1147.784,E2 -1147.784} C_VEL
LIN {X 0,Y 594.638,Z 304.378,A -85,B 0,C 180,E1 -1150.898,E2 -1150.898} C_VEL
LIN {X 0,Y 594.514,Z 324.773,A -85,B 0,C 180,E1 -1153.695,E2 -1153.695} C_VEL
LIN {X 0,Y 594.439,Z 345.484,A -85,B 0,C 180,E1 -1156.497,E2 -1156.497} C_VEL
LIN {X 0,Y 594.441,Z 346.617,A -85,B 0,C 180,E1 -1156.65,E2 -1156.65} C_VEL
LIN {X 0,Y 594.776,Z 350.765,A -85,B 0,C 180,E1 -1156.722,E2 -1156.722} C_VEL
LIN {X 0,Y 594.645,Z 454.975,A -85,B 0,C 180,E1 -1157.999,E2 -1157.999} C_VEL
LIN {X 0,Y 594.62,Z 468.237,A -85,B 0,C 180,E1 -1158.301,E2 -1158.301} C_VEL
LIN {X 0,Y 594.594,Z 480.45,A -85,B 0,C 180,E1 -1158.714,E2 -1158.714} C_VEL
LIN {X 0,Y 594.533,Z 492.642,A -85,B 0,C 180,E1 -1159.271,E2 -1159.271} C_VEL
LIN {X 0,Y 594.46,Z 504.208,A -85,B 0,C 180,E1 -1159.958,E2 -1159.958} C_VEL
LIN {X 0,Y 594.413,Z 514.603,A -85,B 0,C 180,E1 -1160.73,E2 -1160.73} C_VEL
LIN {X 0,Y 594.349,Z 523.034,A -85,B 0,C 180,E1 -1161.501,E2 -1161.501} C_VEL
LIN {X 0,Y 594.347,Z 530.964,A -85,B 0,C 180,E1 -1162.356,E2 -1162.356} C_VEL
LIN {X 0,Y 594.28,Z 538.827,A -85,B 0,C 180,E1 -1163.41,E2 -1163.41} C_VEL
LIN {X 0,Y 594.289,Z 545.683,A -85,B 0,C 180,E1 -1164.572,E2 -1164.572} C_VEL
LIN {X 0,Y 594.27,Z 550.373,A -85,B 0,C 180,E1 -1165.592,E2 -1165.592} C_VEL
LIN {X 0,Y 594.267,Z 553.958,A -85,B 0,C 180,E1 -1166.61,E2 -1166.61} C_VEL
LIN {X 0,Y 594.226,Z 555.81,A -85,B 0,C 180,E1 -1167.289,E2 -1167.289} C_VEL
LIN {X 0,Y 594.24,Z 557.202,A -85,B 0,C 180,E1 -1167.967,E2 -1167.967} C_VEL
LIN {X 0,Y 594.239,Z 558.784,A -85,B 0,C 180,E1 -1169.323,E2 -1169.323} C_VEL
LIN {X 0,Y 594.236,Z 559,A -85,B 0,C 180,E1 -1170,E2 -1170} C_VEL
LIN {X 0,Y 594.247,Z 558.185,A -85,B 0,C 180,E1 -1171.356,E2 -1171.356} C_VEL
LIN {X 0,Y 594.24,Z 557.201,A -85,B 0,C 180,E1 -1172.034,E2 -1172.034} C_VEL
LIN {X 0,Y 594.226,Z 555.809,A -85,B 0,C 180,E1 -1172.712,E2 -1172.712} C_VEL
LIN {X 0,Y 594.288,Z 552.895,A -85,B 0,C 180,E1 -1173.73,E2 -1173.73} C_VEL
LIN {X 0,Y 594.241,Z 548.948,A -85,B 0,C 180,E1 -1174.749,E2 -1174.749} C_VEL
LIN {X 0,Y 594.304,Z 542.876,A -85,B 0,C 180,E1 -1175.94,E2 -1175.94} C_VEL
LIN {X 0,Y 594.308,Z 536.234,A -85,B 0,C 180,E1 -1176.962,E2 -1176.962} C_VEL
LIN {X 0,Y 594.359,Z 527.987,A -85,B 0,C 180,E1 -1177.987,E2 -1177.987} C_VEL
LIN {X 0,Y 594.404,Z 517.597,A -85,B 0,C 180,E1 -1179.013,E2 -1179.013} C_VEL
LIN {X 0,Y 594.448,Z 506.744,A -85,B 0,C 180,E1 -1179.871,E2 -1179.871} C_VEL
LIN {X 0,Y 594.505,Z 495.774,A -85,B 0,C 180,E1 -1180.558,E2 -1180.558} C_VEL
LIN {X 0,Y 594.566,Z 483.558,A -85,B 0,C 180,E1 -1181.159,E2 -1181.159} C_VEL
LIN {X 0,Y 594.565,Z 471.869,A -85,B 0,C 180,E1 -1181.593,E2 -1181.593} C_VEL
LIN {X 0,Y 594.634,Z 459.499,A -85,B 0,C 180,E1 -1181.915,E2 -1181.915} C_VEL
LIN {X 0,Y 594.689,Z 443.716,A -85,B 0,C 180,E1 -1182.152,E2 -1182.152} C_VEL
LIN {X 0,Y 594.622,Z 348.246,A -85,B 0,C 180,E1 -1183.312,E2 -1183.312} C_VEL
LIN {X 0,Y 594.442,Z 346.611,A -85,B 0,C 180,E1 -1183.351,E2 -1183.351} C_VEL
LIN {X 0,Y 594.498,Z 326.062,A -85,B 0,C 180,E1 -1186.13,E2 -1186.13} C_VEL
LIN {X 0,Y 594.607,Z 306.006,A -85,B 0,C 180,E1 -1188.877,E2 -1188.877} C_VEL
LIN {X 0,Y 594.773,Z 283.345,A -85,B 0,C 180,E1 -1192.035,E2 -1192.035} C_VEL
LIN {X 0,Y 594.666,Z 277.938,A -85,B 0,C 180,E1 -1192.804,E2 -1192.804} C_VEL
LIN {X 0,Y 594.392,Z 276.444,A -85,B 0,C 180,E1 -1193.058,E2 -1193.058} C_VEL
LIN {X 0,Y 594.364,Z 276.443,A -85,B 0,C 180,E1 -1195.194,E2 -1195.194} C_VEL
LIN {X 0,Y 594.37,Z 276.444,A -85,B 0,C 180,E1 -1197.523,E2 -1197.523} C_VEL
LIN {X 0,Y 594.388,Z 276.447,A -85,B 0,C 180,E1 -1200.328,E2 -1200.328} C_VEL
LIN {X 0,Y 594.378,Z 276.44,A -85,B 0,C 180,E1 -1202.95,E2 -1202.95} C_VEL
LIN {X 0,Y 594.349,Z 276.444,A -85,B 0,C 180,E1 -1205.409,E2 -1205.409} C_VEL
LIN {X 0,Y 594.383,Z 276.443,A -85,B 0,C 180,E1 -1207.941,E2 -1207.941} C_VEL
LIN {X 0,Y 594.377,Z 276.445,A -85,B 0,C 180,E1 -1210.822,E2 -1210.822} C_VEL
LIN {X 0,Y 594.366,Z 276.442,A -85,B 0,C 180,E1 -1213.299,E2 -1213.299} C_VEL
LIN {X 0,Y 594.36,Z 276.445,A -85,B 0,C 180,E1 -1216.161,E2 -1216.161} C_VEL
LIN {X 0,Y 594.379,Z 276.448,A -85,B 0,C 180,E1 -1218.536,E2 -1218.536} C_VEL
LIN {X 0,Y 594.382,Z 276.442,A -85,B 0,C 180,E1 -1221.296,E2 -1221.296} C_VEL
LIN {X 0,Y 594.351,Z 276.443,A -85,B 0,C 180,E1 -1223.755,E2 -1223.755} C_VEL
LIN {X 0,Y 594.374,Z 276.441,A -85,B 0,C 180,E1 -1226.238,E2 -1226.238} C_VEL
LIN {X 0,Y 594.368,Z 276.446,A -85,B 0,C 180,E1 -1228.649,E2 -1228.649} C_VEL
LIN {X 0,Y 594.381,Z 276.45,A -85,B 0,C 180,E1 -1231.042,E2 -1231.042} C_VEL
LIN {X 0,Y 594.384,Z 276.439,A -85,B 0,C 180,E1 -1233.977,E2 -1233.977} C_VEL
LIN {X 0,Y 594.387,Z 276.438,A -85,B 0,C 180,E1 -1236.296,E2 -1236.296} C_VEL
LIN {X 0,Y 594.403,Z 276.445,A -85,B 0,C 180,E1 -1239.224,E2 -1239.224} C_VEL
LIN {X 0,Y 594.35,Z 276.444,A -85,B 0,C 180,E1 -1242.095,E2 -1242.095} C_VEL
LIN {X 0,Y 594.363,Z 276.442,A -85,B 0,C 180,E1 -1244.219,E2 -1244.219} C_VEL
LIN {X 0,Y 594.378,Z 276.44,A -85,B 0,C 180,E1 -1246.321,E2 -1246.321} C_VEL
LIN {X 0,Y 594.371,Z 276.442,A -85,B 0,C 180,E1 -1249.094,E2 -1249.094} C_VEL
LIN {X 0,Y 594.409,Z 276.445,A -85,B 0,C 180,E1 -1251.843,E2 -1251.843} C_VEL
LIN {X 0,Y 594.393,Z 276.438,A -85,B 0,C 180,E1 -1254.572,E2 -1254.572} C_VEL
LIN {X 0,Y 594.4,Z 276.438,A -85,B 0,C 180,E1 -1257.289,E2 -1257.289} C_VEL
LIN {X 0,Y 594.413,Z 276.446,A -85,B 0,C 180,E1 -1260,E2 -1260} C_VEL
LIN {X 0,Y 594.401,Z 276.438,A -85,B 0,C 180,E1 -1262.711,E2 -1262.711} C_VEL
LIN {X 0,Y 594.392,Z 276.438,A -85,B 0,C 180,E1 -1265.428,E2 -1265.428} C_VEL
LIN {X 0,Y 594.408,Z 276.445,A -85,B 0,C 180,E1 -1268.157,E2 -1268.157} C_VEL
LIN {X 0,Y 594.386,Z 276.439,A -85,B 0,C 180,E1 -1271.074,E2 -1271.074} C_VEL
LIN {X 0,Y 594.379,Z 276.44,A -85,B 0,C 180,E1 -1273.679,E2 -1273.679} C_VEL
LIN {X 0,Y 594.358,Z 276.442,A -85,B 0,C 180,E1 -1275.321,E2 -1275.321} C_VEL
LIN {X 0,Y 593.682,Z 276.529,A -85,B 0,C 180,E1 -1275.886,E2 -1275.886} C_VEL
LIN {X 0,Y 590.816,Z 276.89,A -85,B 0,C 180,E1 -1276.804,E2 -1276.804} C_VEL
LIN {X 0,Y 588.406,Z 277.189,A -85,B 0,C 180,E1 -1277.543,E2 -1277.543} C_VEL
LIN {X 0,Y 587.385,Z 277.314,A -85,B 0,C 180,E1 -1278.113,E2 -1278.113} C_VEL
LIN {X 0,Y 587.308,Z 277.324,A -85,B 0,C 180,E1 -1278.306,E2 -1278.306} C_VEL
LIN {X 0,Y 587.328,Z 277.323,A -85,B 0,C 180,E1 -1281.038,E2 -1281.038} C_VEL
LIN {X 0,Y 587.321,Z 277.321,A -85,B 0,C 180,E1 -1283.259,E2 -1283.259} C_VEL
LIN {X 0,Y 587.332,Z 277.318,A -85,B 0,C 180,E1 -1285.517,E2 -1285.517} C_VEL
LIN {X 0,Y 587.344,Z 277.315,A -85,B 0,C 180,E1 -1287.818,E2 -1287.818} C_VEL
LIN {X 0,Y 587.335,Z 277.32,A -85,B 0,C 180,E1 -1290.51,E2 -1290.51} C_VEL
LIN {X 0,Y 587.331,Z 277.323,A -85,B 0,C 180,E1 -1293.397,E2 -1293.397} C_VEL
LIN {X 0,Y 587.289,Z 277.323,A -85,B 0,C 180,E1 -1295.9,E2 -1295.9} C_VEL
LIN {X 0,Y 587.328,Z 277.319,A -85,B 0,C 180,E1 -1298.48,E2 -1298.48} C_VEL
LIN {X 0,Y 587.335,Z 277.325,A -85,B 0,C 180,E1 -1301.157,E2 -1301.157} C_VEL
LIN {X 0,Y 587.311,Z 277.321,A -85,B 0,C 180,E1 -1304.112,E2 -1304.112} C_VEL
LIN {X 0,Y 587.313,Z 277.323,A -85,B 0,C 180,E1 -1306.994,E2 -1306.994} C_VEL
LIN {X 0,Y 587.311,Z 277.329,A -85,B 0,C 180,E1 -1309.746,E2 -1309.746} C_VEL
LIN {X 0,Y 587.344,Z 277.317,A -85,B 0,C 180,E1 -1312.392,E2 -1312.392} C_VEL
LIN {X 0,Y 587.341,Z 277.326,A -85,B 0,C 180,E1 -1315.653,E2 -1315.653} C_VEL
LIN {X 0,Y 587.34,Z 277.322,A -85,B 0,C 180,E1 -1318.231,E2 -1318.231} C_VEL
LIN {X 0,Y 587.362,Z 277.451,A -85,B 0,C 180,E1 -1321.11,E2 -1321.11} C_VEL
LIN {X 0,Y 587.44,Z 288.921,A -85,B 0,C 180,E1 -1323.152,E2 -1323.152} C_VEL
LIN {X 0,Y 587.373,Z 303.485,A -85,B 0,C 180,E1 -1325.707,E2 -1325.707} C_VEL
LIN {X 0,Y 587.299,Z 308.402,A -85,B 0,C 180,E1 -1326.562,E2 -1326.562} C_VEL
LIN {X 0,Y 587.897,Z 313.638,A -85,B 0,C 180,E1 -1326.645,E2 -1326.645} C_VEL
LIN {X 0,Y 587.687,Z 414.639,A -85,B 0,C 180,E1 -1327.894,E2 -1327.894} C_VEL
LIN {X 0,Y 587.598,Z 427.74,A -85,B 0,C 180,E1 -1328.19,E2 -1328.19} C_VEL
LIN {X 0,Y 587.577,Z 439.989,A -85,B 0,C 180,E1 -1328.604,E2 -1328.604} C_VEL
LIN {X 0,Y 587.532,Z 452.027,A -85,B 0,C 180,E1 -1329.153,E2 -1329.153} C_VEL
LIN {X 0,Y 587.447,Z 462.863,A -85,B 0,C 180,E1 -1329.791,E2 -1329.791} C_VEL
LIN {X 0,Y 587.389,Z 473.618,A -85,B 0,C 180,E1 -1330.582,E2 -1330.582} C_VEL
LIN {X 0,Y 587.347,Z 481.958,A -85,B 0,C 180,E1 -1331.332,E2 -1331.332} C_VEL
LIN {X 0,Y 587.306,Z 490.318,A -85,B 0,C 180,E1 -1332.233,E2 -1332.233} C_VEL
LIN {X 0,Y 587.254,Z 498.386,A -85,B 0,C 180,E1 -1333.308,E2 -1333.308} C_VEL
LIN {X 0,Y 587.196,Z 504.77,A -85,B 0,C 180,E1 -1334.377,E2 -1334.377} C_VEL
LIN {X 0,Y 587.189,Z 509.791,A -85,B 0,C 180,E1 -1335.443,E2 -1335.443} C_VEL
LIN {X 0,Y 587.16,Z 513.614,A -85,B 0,C 180,E1 -1336.502,E2 -1336.502} C_VEL
LIN {X 0,Y 587.162,Z 516.362,A -85,B 0,C 180,E1 -1337.558,E2 -1337.558} C_VEL
LIN {X 0,Y 587.154,Z 517.639,A -85,B 0,C 180,E1 -1338.259,E2 -1338.259} C_VEL
LIN {X 0,Y 587.165,Z 518.504,A -85,B 0,C 180,E1 -1338.959,E2 -1338.959} C_VEL
LIN {X 0,Y 587.15,Z 518.936,A -85,B 0,C 180,E1 -1340.353,E2 -1340.353} C_VEL
LIN {X 0,Y 587.127,Z 518.567,A -85,B 0,C 180,E1 -1341.047,E2 -1341.047} C_VEL
LIN {X 0,Y 587.137,Z 517.782,A -85,B 0,C 180,E1 -1341.741,E2 -1341.741} C_VEL
LIN {X 0,Y 587.145,Z 516.566,A -85,B 0,C 180,E1 -1342.434,E2 -1342.434} C_VEL
LIN {X 0,Y 587.194,Z 514.134,A -85,B 0,C 180,E1 -1343.418,E2 -1343.418} C_VEL
LIN {X 0,Y 587.189,Z 510.379,A -85,B 0,C 180,E1 -1344.505,E2 -1344.505} C_VEL
LIN {X 0,Y 587.198,Z 505.689,A -85,B 0,C 180,E1 -1345.538,E2 -1345.538} C_VEL
LIN {X 0,Y 587.214,Z 498.656,A -85,B 0,C 180,E1 -1346.741,E2 -1346.741} C_VEL
LIN {X 0,Y 587.256,Z 491.059,A -85,B 0,C 180,E1 -1347.771,E2 -1347.771} C_VEL
LIN {X 0,Y 587.346,Z 481.546,A -85,B 0,C 180,E1 -1348.8,E2 -1348.8} C_VEL
LIN {X 0,Y 587.39,Z 471.787,A -85,B 0,C 180,E1 -1349.657,E2 -1349.657} C_VEL
LIN {X 0,Y 587.45,Z 460.853,A -85,B 0,C 180,E1 -1350.428,E2 -1350.428} C_VEL
LIN {X 0,Y 587.543,Z 448.478,A -85,B 0,C 180,E1 -1351.113,E2 -1351.113} C_VEL
LIN {X 0,Y 587.63,Z 436.281,A -85,B 0,C 180,E1 -1351.627,E2 -1351.627} C_VEL
LIN {X 0,Y 587.644,Z 423.417,A -85,B 0,C 180,E1 -1352.013,E2 -1352.013} C_VEL
LIN {X 0,Y 587.731,Z 409.626,A -85,B 0,C 180,E1 -1352.27,E2 -1352.27} C_VEL
LIN {X 0,Y 587.745,Z 311.049,A -85,B 0,C 180,E1 -1353.481,E2 -1353.481} C_VEL
LIN {X 0,Y 587.281,Z 308.349,A -85,B 0,C 180,E1 -1353.537,E2 -1353.537} C_VEL
LIN {X 0,Y 587.333,Z 297.148,A -85,B 0,C 180,E1 -1355.493,E2 -1355.493} C_VEL
LIN {X 0,Y 587.501,Z 281.5,A -85,B 0,C 180,E1 -1358.253,E2 -1358.253} C_VEL
LIN {X 0,Y 587.31,Z 277.325,A -85,B 0,C 180,E1 -1359.036,E2 -1359.036} C_VEL
LIN {X 0,Y 587.302,Z 277.325,A -85,B 0,C 180,E1 -1361.737,E2 -1361.737} C_VEL
LIN {X 0,Y 587.328,Z 277.324,A -85,B 0,C 180,E1 -1364.553,E2 -1364.553} C_VEL
LIN {X 0,Y 587.277,Z 277.324,A -85,B 0,C 180,E1 -1367.408,E2 -1367.408} C_VEL
LIN {X 0,Y 587.294,Z 277.322,A -85,B 0,C 180,E1 -1369.576,E2 -1369.576} C_VEL
LIN {X 0,Y 587.301,Z 277.322,A -85,B 0,C 180,E1 -1371.774,E2 -1371.774} C_VEL
LIN {X 0,Y 587.295,Z 277.33,A -85,B 0,C 180,E1 -1374.76,E2 -1374.76} C_VEL
LIN {X 0,Y 587.294,Z 277.322,A -85,B 0,C 180,E1 -1377.682,E2 -1377.682} C_VEL
LIN {X 0,Y 587.29,Z 277.325,A -85,B 0,C 180,E1 -1380.172,E2 -1380.172} C_VEL
LIN {X 0,Y 587.325,Z 277.326,A -85,B 0,C 180,E1 -1382.579,E2 -1382.579} C_VEL
LIN {X 0,Y 587.318,Z 277.327,A -85,B 0,C 180,E1 -1385.055,E2 -1385.055} C_VEL
LIN {X 0,Y 587.322,Z 277.319,A -85,B 0,C 180,E1 -1387.836,E2 -1387.836} C_VEL
LIN {X 0,Y 587.299,Z 277.322,A -85,B 0,C 180,E1 -1390.254,E2 -1390.254} C_VEL
LIN {X 0,Y 587.296,Z 277.332,A -85,B 0,C 180,E1 -1393.116,E2 -1393.116} C_VEL
LIN {X 0,Y 587.29,Z 277.323,A -85,B 0,C 180,E1 -1396.046,E2 -1396.046} C_VEL
LIN {X 0,Y 587.323,Z 277.324,A -85,B 0,C 180,E1 -1398.925,E2 -1398.925} C_VEL
LIN {X 0,Y 587.318,Z 277.326,A -85,B 0,C 180,E1 -1401.52,E2 -1401.52} C_VEL
LIN {X 0,Y 587.281,Z 277.325,A -85,B 0,C 180,E1 -1404.099,E2 -1404.099} C_VEL
LIN {X 0,Y 587.319,Z 277.319,A -85,B 0,C 180,E1 -1406.602,E2 -1406.602} C_VEL
LIN {X 0,Y 587.326,Z 277.33,A -85,B 0,C 180,E1 -1409.49,E2 -1409.49} C_VEL
LIN {X 0,Y 587.297,Z 277.324,A -85,B 0,C 180,E1 -1412.18,E2 -1412.18} C_VEL
LIN {X 0,Y 587.321,Z 277.319,A -85,B 0,C 180,E1 -1414.483,E2 -1414.483} C_VEL
LIN {X 0,Y 587.329,Z 277.325,A -85,B 0,C 180,E1 -1417.486,E2 -1417.486} C_VEL
LIN {X 0,Y 587.304,Z 277.323,A -85,B 0,C 180,E1 -1420.424,E2 -1420.424} C_VEL
LIN {X 0,Y 587.318,Z 277.322,A -85,B 0,C 180,E1 -1423.31,E2 -1423.31} C_VEL
LIN {X 0,Y 587.35,Z 277.323,A -85,B 0,C 180,E1 -1426.154,E2 -1426.154} C_VEL
LIN {X 0,Y 587.326,Z 277.318,A -85,B 0,C 180,E1 -1428.962,E2 -1428.962} C_VEL
LIN {X 0,Y 587.355,Z 277.32,A -85,B 0,C 180,E1 -1431.745,E2 -1431.745} C_VEL
LIN {X 0,Y 587.358,Z 277.319,A -85,B 0,C 180,E1 -1434.507,E2 -1434.507} C_VEL
LIN {X 0,Y 587.358,Z 277.314,A -85,B 0,C 180,E1 -1437.257,E2 -1437.257} C_VEL
LIN {X 0,Y 587.368,Z 277.318,A -85,B 0,C 180,E1 -1440,E2 -1440} C_VEL
LIN {X 0,Y 587.373,Z 277.317,A -85,B 0,C 180,E1 -1442.743,E2 -1442.743} C_VEL
LIN {X 0,Y 587.35,Z 277.315,A -85,B 0,C 180,E1 -1445.493,E2 -1445.493} C_VEL
LIN {X 0,Y 587.36,Z 277.32,A -85,B 0,C 180,E1 -1448.255,E2 -1448.255} C_VEL
LIN {X 0,Y 587.354,Z 277.317,A -85,B 0,C 180,E1 -1451.142,E2 -1451.142} C_VEL
LIN {X 0,Y 587.355,Z 277.318,A -85,B 0,C 180,E1 -1454.261,E2 -1454.261} C_VEL
LIN {X 0,Y 587.343,Z 277.318,A -85,B 0,C 180,E1 -1457.406,E2 -1457.406} C_VEL
LIN {X 0,Y 587.321,Z 277.321,A -85,B 0,C 180,E1 -1460.305,E2 -1460.305} C_VEL
LIN {X 0,Y 587.316,Z 277.325,A -85,B 0,C 180,E1 -1463.259,E2 -1463.259} C_VEL
LIN {X 0,Y 587.331,Z 277.32,A -85,B 0,C 180,E1 -1465.517,E2 -1465.517} C_VEL
LIN {X 0,Y 587.341,Z 277.317,A -85,B 0,C 180,E1 -1467.818,E2 -1467.818} C_VEL
LIN {X 0,Y 587.344,Z 277.318,A -85,B 0,C 180,E1 -1470.513,E2 -1470.513} C_VEL
LIN {X 0,Y 587.329,Z 277.325,A -85,B 0,C 180,E1 -1473.397,E2 -1473.397} C_VEL
LIN {X 0,Y 587.313,Z 277.322,A -85,B 0,C 180,E1 -1475.899,E2 -1475.899} C_VEL
LIN {X 0,Y 587.327,Z 277.318,A -85,B 0,C 180,E1 -1478.48,E2 -1478.48} C_VEL
LIN {X 0,Y 587.332,Z 277.324,A -85,B 0,C 180,E1 -1481.158,E2 -1481.158} C_VEL
LIN {X 0,Y 587.322,Z 277.32,A -85,B 0,C 180,E1 -1484.114,E2 -1484.114} C_VEL
LIN {X 0,Y 587.312,Z 277.322,A -85,B 0,C 180,E1 -1486.995,E2 -1486.995} C_VEL
LIN {X 0,Y 587.31,Z 277.33,A -85,B 0,C 180,E1 -1489.746,E2 -1489.746} C_VEL
LIN {X 0,Y 587.343,Z 277.317,A -85,B 0,C 180,E1 -1492.393,E2 -1492.393} C_VEL
LIN {X 0,Y 587.359,Z 277.325,A -85,B 0,C 180,E1 -1495.781,E2 -1495.781} C_VEL
LIN {X 0,Y 587.339,Z 277.321,A -85,B 0,C 180,E1 -1498.232,E2 -1498.232} C_VEL
LIN {X 0,Y 587.348,Z 277.316,A -85,B 0,C 180,E1 -1500.867,E2 -1500.867} C_VEL
LIN {X 0,Y 587.357,Z 277.323,A -85,B 0,C 180,E1 -1503.82,E2 -1503.82} C_VEL
LIN {X 0,Y 587.337,Z 277.324,A -85,B 0,C 180,E1 -1506.743,E2 -1506.743} C_VEL
LIN {X 0,Y 587.378,Z 277.604,A -85,B 0,C 180,E1 -1506.849,E2 -1506.849} C_VEL
LIN {X 0,Y 587.867,Z 282.056,A -85,B 0,C 180,E1 -1507.508,E2 -1507.508} C_VEL
LIN {X 0,Y 587.705,Z 302.767,A -85,B 0,C 180,E1 -1510.438,E2 -1510.438} C_VEL
LIN {X 0,Y 587.55,Z 322.066,A -85,B 0,C 180,E1 -1513.122,E2 -1513.122} C_VEL
LIN {X 0,Y 587.428,Z 344.19,A -85,B 0,C 180,E1 -1516.157,E2 -1516.157} C_VEL
LIN {X 0,Y 587.392,Z 346.617,A -85,B 0,C 180,E1 -1516.486,E2 -1516.486} C_VEL
LIN {X 0,Y 587.869,Z 350.765,A -85,B 0,C 180,E1 -1516.564,E2 -1516.564} C_VEL
LIN {X 0,Y 587.724,Z 454.975,A -85,B 0,C 180,E1 -1517.856,E2 -1517.856} C_VEL
LIN {X 0,Y 587.671,Z 468.238,A -85,B 0,C 180,E1 -1518.161,E2 -1518.161} C_VEL
LIN {X 0,Y 587.624,Z 480.655,A -85,B 0,C 180,E1 -1518.586,E2 -1518.586} C_VEL
LIN {X 0,Y 587.555,Z 492.64,A -85,B 0,C 180,E1 -1519.142,E2 -1519.142} C_VEL
LIN {X 0,Y 587.442,Z 504.209,A -85,B 0,C 180,E1 -1519.837,E2 -1519.837} C_VEL
LIN {X 0,Y 587.392,Z 514.604,A -85,B 0,C 180,E1 -1520.618,E2 -1520.618} C_VEL
LIN {X 0,Y 587.299,Z 523.047,A -85,B 0,C 180,E1 -1521.398,E2 -1521.398} C_VEL
LIN {X 0,Y 587.273,Z 530.964,A -85,B 0,C 180,E1 -1522.263,E2 -1522.263} C_VEL
LIN {X 0,Y 587.229,Z 537.472,A -85,B 0,C 180,E1 -1523.127,E2 -1523.127} C_VEL
LIN {X 0,Y 587.236,Z 543.869,A -85,B 0,C 180,E1 -1524.162,E2 -1524.162} C_VEL
LIN {X 0,Y 587.147,Z 548.952,A -85,B 0,C 180,E1 -1525.194,E2 -1525.194} C_VEL
LIN {X 0,Y 587.212,Z 552.897,A -85,B 0,C 180,E1 -1526.226,E2 -1526.226} C_VEL
LIN {X 0,Y 587.132,Z 555.81,A -85,B 0,C 180,E1 -1527.256,E2 -1527.256} C_VEL
LIN {X 0,Y 587.139,Z 557.201,A -85,B 0,C 180,E1 -1527.942,E2 -1527.942} C_VEL
LIN {X 0,Y 587.14,Z 558.785,A -85,B 0,C 180,E1 -1529.315,E2 -1529.315} C_VEL
LIN {X 0,Y 587.137,Z 559,A -85,B 0,C 180,E1 -1530,E2 -1530} C_VEL
LIN {X 0,Y 587.147,Z 558.185,A -85,B 0,C 180,E1 -1531.372,E2 -1531.372} C_VEL
LIN {X 0,Y 587.139,Z 557.2,A -85,B 0,C 180,E1 -1532.058,E2 -1532.058} C_VEL
LIN {X 0,Y 587.132,Z 555.809,A -85,B 0,C 180,E1 -1532.745,E2 -1532.745} C_VEL
LIN {X 0,Y 587.212,Z 552.895,A -85,B 0,C 180,E1 -1533.775,E2 -1533.775} C_VEL
LIN {X 0,Y 587.147,Z 548.948,A -85,B 0,C 180,E1 -1534.807,E2 -1534.807} C_VEL
LIN {X 0,Y 587.217,Z 542.876,A -85,B 0,C 180,E1 -1536.011,E2 -1536.011} C_VEL
LIN {X 0,Y 587.245,Z 536.235,A -85,B 0,C 180,E1 -1537.046,E2 -1537.046} C_VEL
LIN {X 0,Y 587.297,Z 527.988,A -85,B 0,C 180,E1 -1538.083,E2 -1538.083} C_VEL
LIN {X 0,Y 587.357,Z 517.598,A -85,B 0,C 180,E1 -1539.123,E2 -1539.123} C_VEL
LIN {X 0,Y 587.444,Z 506.744,A -85,B 0,C 180,E1 -1539.99,E2 -1539.99} C_VEL
LIN {X 0,Y 587.521,Z 495.776,A -85,B 0,C 180,E1 -1540.685,E2 -1540.685} C_VEL
LIN {X 0,Y 587.602,Z 483.792,A -85,B 0,C 180,E1 -1541.282,E2 -1541.282} C_VEL
LIN {X 0,Y 587.618,Z 471.867,A -85,B 0,C 180,E1 -1541.732,E2 -1541.732} C_VEL
LIN {X 0,Y 587.689,Z 459.497,A -85,B 0,C 180,E1 -1542.058,E2 -1542.058} C_VEL
LIN {X 0,Y 587.744,Z 443.716,A -85,B 0,C 180,E1 -1542.298,E2 -1542.298} C_VEL
LIN {X 0,Y 587.716,Z 348.814,A -85,B 0,C 180,E1 -1543.464,E2 -1543.464} C_VEL
LIN {X 0,Y 587.392,Z 346.611,A -85,B 0,C 180,E1 -1543.514,E2 -1543.514} C_VEL
LIN {X 0,Y 587.47,Z 328.651,A -85,B 0,C 180,E1 -1545.971,E2 -1545.971} C_VEL
LIN {X 0,Y 587.632,Z 309.234,A -85,B 0,C 180,E1 -1548.659,E2 -1548.659} C_VEL
LIN {X 0,Y 587.802,Z 288.498,A -85,B 0,C 180,E1 -1551.575,E2 -1551.575} C_VEL
LIN {X 0,Y 587.805,Z 279.778,A -85,B 0,C 180,E1 -1552.821,E2 -1552.821} C_VEL
LIN {X 0,Y 587.335,Z 277.325,A -85,B 0,C 180,E1 -1553.206,E2 -1553.206} C_VEL
LIN {X 0,Y 587.326,Z 277.323,A -85,B 0,C 180,E1 -1555.517,E2 -1555.517} C_VEL
LIN {X 0,Y 587.342,Z 277.324,A -85,B 0,C 180,E1 -1557.818,E2 -1557.818} C_VEL
LIN {X 0,Y 587.339,Z 277.322,A -85,B 0,C 180,E1 -1560.51,E2 -1560.51} C_VEL
LIN {X 0,Y 587.329,Z 277.318,A -85,B 0,C 180,E1 -1563.397,E2 -1563.397} C_VEL
LIN {X 0,Y 587.291,Z 277.327,A -85,B 0,C 180,E1 -1565.9,E2 -1565.9} C_VEL
LIN {X 0,Y 587.327,Z 277.328,A -85,B 0,C 180,E1 -1568.479,E2 -1568.479} C_VEL
LIN {X 0,Y 587.336,Z 277.318,A -85,B 0,C 180,E1 -1571.157,E2 -1571.157} C_VEL
LIN {X 0,Y 587.312,Z 277.324,A -85,B 0,C 180,E1 -1574.112,E2 -1574.112} C_VEL
LIN {X 0,Y 587.316,Z 277.325,A -85,B 0,C 180,E1 -1576.993,E2 -1576.993} C_VEL
LIN {X 0,Y 587.312,Z 277.32,A -85,B 0,C 180,E1 -1579.745,E2 -1579.745} C_VEL
LIN {X 0,Y 587.345,Z 277.32,A -85,B 0,C 180,E1 -1582.392,E2 -1582.392} C_VEL
LIN {X 0,Y 587.36,Z 277.314,A -85,B 0,C 180,E1 -1585.78,E2 -1585.78} C_VEL
LIN {X 0,Y 587.339,Z 277.317,A -85,B 0,C 180,E1 -1588.231,E2 -1588.231} C_VEL
LIN {X 0,Y 587.348,Z 277.322,A -85,B 0,C 180,E1 -1590.866,E2 -1590.866} C_VEL
LIN {X 0,Y 587.358,Z 277.316,A -85,B 0,C 180,E1 -1593.819,E2 -1593.819} C_VEL
LIN {X 0,Y 587.335,Z 277.318,A -85,B 0,C 180,E1 -1595.993,E2 -1595.993} C_VEL
LIN {X 0,Y 587.319,Z 277.319,A -85,B 0,C 180,E1 -1598.225,E2 -1598.225} C_VEL
LIN {X 0,Y 587.35,Z 277.321,A -85,B 0,C 180,E1 -1601.151,E2 -1601.151} C_VEL
LIN {X 0,Y 587.321,Z 277.321,A -85,B 0,C 180,E1 -1604.025,E2 -1604.025} C_VEL
LIN {X 0,Y 587.356,Z 277.316,A -85,B 0,C 180,E1 -1606.154,E2 -1606.154} C_VEL
LIN {X 0,Y 587.337,Z 277.317,A -85,B 0,C 180,E1 -1608.962,E2 -1608.962} C_VEL
LIN {X 0,Y 587.362,Z 277.325,A -85,B 0,C 180,E1 -1611.745,E2 -1611.745} C_VEL
LIN {X 0,Y 587.357,Z 277.315,A -85,B 0,C 180,E1 -1614.507,E2 -1614.507} C_VEL
LIN {X 0,Y 587.367,Z 277.314,A -85,B 0,C 180,E1 -1617.257,E2 -1617.257} C_VEL
LIN {X 0,Y 587.382,Z 277.322,A -85,B 0,C 180,E1 -1620,E2 -1620} C_VEL
LIN {X 0,Y 587.368,Z 277.314,A -85,B 0,C 180,E1 -1622.743,E2 -1622.743} C_VEL
LIN {X 0,Y 587.356,Z 277.315,A -85,B 0,C 180,E1 -1625.493,E2 -1625.493} C_VEL
LIN {X 0,Y 587.361,Z 277.324,A -85,B 0,C 180,E1 -1628.255,E2 -1628.255} C_VEL
LIN {X 0,Y 587.345,Z 277.316,A -85,B 0,C 180,E1 -1631.134,E2 -1631.134} C_VEL
LIN {X 0,Y 587.362,Z 277.321,A -85,B 0,C 180,E1 -1634.26,E2 -1634.26} C_VEL
LIN {X 0,Y 587.346,Z 277.316,A -85,B 0,C 180,E1 -1637.406,E2 -1637.406} C_VEL
LIN {X 0,Y 587.308,Z 277.324,A -85,B 0,C 180,E1 -1638.306,E2 -1638.306} C_VEL
LIN {X 0,Y 586.666,Z 277.408,A -85,B 0,C 180,E1 -1638.878,E2 -1638.878} C_VEL
LIN {X 0,Y 583.841,Z 277.759,A -85,B 0,C 180,E1 -1639.807,E2 -1639.807} C_VEL
LIN {X 0,Y 581.43,Z 278.062,A -85,B 0,C 180,E1 -1640.554,E2 -1640.554} C_VEL
LIN {X 0,Y 580.376,Z 278.188,A -85,B 0,C 180,E1 -1641.13,E2 -1641.13} C_VEL
LIN {X 0,Y 580.281,Z 278.197,A -85,B 0,C 180,E1 -1641.325,E2 -1641.325} C_VEL
LIN {X 0,Y 580.278,Z 278.196,A -85,B 0,C 180,E1 -1643.558,E2 -1643.558} C_VEL
LIN {X 0,Y 580.29,Z 278.194,A -85,B 0,C 180,E1 -1645.849,E2 -1645.849} C_VEL
LIN {X 0,Y 580.296,Z 278.194,A -85,B 0,C 180,E1 -1648.186,E2 -1648.186} C_VEL
LIN {X 0,Y 580.283,Z 278.202,A -85,B 0,C 180,E1 -1650.695,E2 -1650.695} C_VEL
LIN {X 0,Y 580.3,Z 278.2,A -85,B 0,C 180,E1 -1653.316,E2 -1653.316} C_VEL
LIN {X 0,Y 580.244,Z 278.202,A -85,B 0,C 180,E1 -1655.756,E2 -1655.756} C_VEL
LIN {X 0,Y 580.287,Z 278.195,A -85,B 0,C 180,E1 -1658.146,E2 -1658.146} C_VEL
LIN {X 0,Y 580.297,Z 278.197,A -85,B 0,C 180,E1 -1660.844,E2 -1660.844} C_VEL
LIN {X 0,Y 580.272,Z 278.203,A -85,B 0,C 180,E1 -1663.659,E2 -1663.659} C_VEL
LIN {X 0,Y 580.273,Z 278.197,A -85,B 0,C 180,E1 -1666.61,E2 -1666.61} C_VEL
LIN {X 0,Y 580.298,Z 278.198,A -85,B 0,C 180,E1 -1669.157,E2 -1669.157} C_VEL
LIN {X 0,Y 580.289,Z 278.201,A -85,B 0,C 180,E1 -1671.927,E2 -1671.927} C_VEL
LIN {X 0,Y 580.25,Z 278.201,A -85,B 0,C 180,E1 -1674.453,E2 -1674.453} C_VEL
LIN {X 0,Y 580.289,Z 278.196,A -85,B 0,C 180,E1 -1676.975,E2 -1676.975} C_VEL
LIN {X 0,Y 580.296,Z 278.199,A -85,B 0,C 180,E1 -1679.425,E2 -1679.425} C_VEL
LIN {X 0,Y 580.331,Z 278.301,A -85,B 0,C 180,E1 -1681.026,E2 -1681.026} C_VEL
LIN {X 0,Y 580.412,Z 288.134,A -85,B 0,C 180,E1 -1682.8,E2 -1682.8} C_VEL
LIN {X 0,Y 580.331,Z 304.365,A -85,B 0,C 180,E1 -1685.685,E2 -1685.685} C_VEL
LIN {X 0,Y 580.251,Z 308.39,A -85,B 0,C 180,E1 -1686.393,E2 -1686.393} C_VEL
LIN {X 0,Y 580.998,Z 314.11,A -85,B 0,C 180,E1 -1686.488,E2 -1686.488} C_VEL
LIN {X 0,Y 580.743,Z 415.141,A -85,B 0,C 180,E1 -1687.756,E2 -1687.756} C_VEL
LIN {X 0,Y 580.644,Z 428.064,A -85,B 0,C 180,E1 -1688.056,E2 -1688.056} C_VEL
LIN {X 0,Y 580.618,Z 441.403,A -85,B 0,C 180,E1 -1688.521,E2 -1688.521} C_VEL
LIN {X 0,Y 580.53,Z 453.319,A -85,B 0,C 180,E1 -1689.092,E2 -1689.092} C_VEL
LIN {X 0,Y 580.41,Z 465.009,A -85,B 0,C 180,E1 -1689.812,E2 -1689.812} C_VEL
LIN {X 0,Y 580.363,Z 475.041,A -85,B 0,C 180,E1 -1690.585,E2 -1690.585} C_VEL
LIN {X 0,Y 580.298,Z 484.273,A -85,B 0,C 180,E1 -1691.463,E2 -1691.463} C_VEL
LIN {X 0,Y 580.205,Z 492.214,A -85,B 0,C 180,E1 -1692.373,E2 -1692.373} C_VEL
LIN {X 0,Y 580.171,Z 499.979,A -85,B 0,C 180,E1 -1693.474,E2 -1693.474} C_VEL
LIN {X 0,Y 580.107,Z 505.985,A -85,B 0,C 180,E1 -1694.542,E2 -1694.542} C_VEL
LIN {X 0,Y 580.087,Z 511.23,A -85,B 0,C 180,E1 -1695.751,E2 -1695.751} C_VEL
LIN {X 0,Y 580.076,Z 514.32,A -85,B 0,C 180,E1 -1696.691,E2 -1696.691} C_VEL
LIN {X 0,Y 580.056,Z 516.103,A -85,B 0,C 180,E1 -1697.403,E2 -1697.403} C_VEL
LIN {X 0,Y 580.054,Z 517.443,A -85,B 0,C 180,E1 -1698.113,E2 -1698.113} C_VEL
LIN {X 0,Y 580.071,Z 518.485,A -85,B 0,C 180,E1 -1698.925,E2 -1698.925} C_VEL
LIN {X 0,Y 580.057,Z 518.964,A -85,B 0,C 180,E1 -1700.234,E2 -1700.234} C_VEL
LIN {X 0,Y 580.059,Z 517.948,A -85,B 0,C 180,E1 -1701.64,E2 -1701.64} C_VEL
LIN {X 0,Y 580.065,Z 516.818,A -85,B 0,C 180,E1 -1702.341,E2 -1702.341} C_VEL
LIN {X 0,Y 580.108,Z 514.229,A -85,B 0,C 180,E1 -1703.429,E2 -1703.429} C_VEL
LIN {X 0,Y 580.111,Z 510.87,A -85,B 0,C 180,E1 -1704.438,E2 -1704.438} C_VEL
LIN {X 0,Y 580.119,Z 506.315,A -85,B 0,C 180,E1 -1705.483,E2 -1705.483} C_VEL
LIN {X 0,Y 580.124,Z 499.439,A -85,B 0,C 180,E1 -1706.701,E2 -1706.701} C_VEL
LIN {X 0,Y 580.197,Z 492.013,A -85,B 0,C 180,E1 -1707.743,E2 -1707.743} C_VEL
LIN {X 0,Y 580.291,Z 484.421,A -85,B 0,C 180,E1 -1708.612,E2 -1708.612} C_VEL
LIN {X 0,Y 580.335,Z 475.358,A -85,B 0,C 180,E1 -1709.479,E2 -1709.479} C_VEL
LIN {X 0,Y 580.398,Z 465.274,A -85,B 0,C 180,E1 -1710.26,E2 -1710.26} C_VEL
LIN {X 0,Y 580.544,Z 454.121,A -85,B 0,C 180,E1 -1710.953,E2 -1710.953} C_VEL
LIN {X 0,Y 580.647,Z 443.58,A -85,B 0,C 180,E1 -1711.473,E2 -1711.473} C_VEL
LIN {X 0,Y 580.683,Z 430.912,A -85,B 0,C 180,E1 -1711.95,E2 -1711.95} C_VEL
LIN {X 0,Y 580.755,Z 418.17,A -85,B 0,C 180,E1 -1712.275,E2 -1712.275} C_VEL
LIN {X 0,Y 580.829,Z 400.218,A -85,B 0,C 180,E1 -1712.535,E2 -1712.535} C_VEL
LIN {X 0,Y 580.82,Z 311.777,A -85,B 0,C 180,E1 -1713.635,E2 -1713.635} C_VEL
LIN {X 0,Y 580.259,Z 308.31,A -85,B 0,C 180,E1 -1713.711,E2 -1713.711} C_VEL
LIN {X 0,Y 580.36,Z 295.885,A -85,B 0,C 180,E1 -1715.908,E2 -1715.908} C_VEL
LIN {X 0,Y 580.456,Z 280.266,A -85,B 0,C 180,E1 -1718.704,E2 -1718.704} C_VEL
LIN {X 0,Y 580.268,Z 278.203,A -85,B 0,C 180,E1 -1719.102,E2 -1719.102} C_VEL
LIN {X 0,Y 580.28,Z 278.202,A -85,B 0,C 180,E1 -1721.881,E2 -1721.881} C_VEL
LIN {X 0,Y 580.276,Z 278.2,A -85,B 0,C 180,E1 -1724.734,E2 -1724.734} C_VEL
LIN {X 0,Y 580.243,Z 278.201,A -85,B 0,C 180,E1 -1727.625,E2 -1727.625} C_VEL
LIN {X 0,Y 580.273,Z 278.198,A -85,B 0,C 180,E1 -1729.823,E2 -1729.823} C_VEL
LIN {X 0,Y 580.255,Z 278.203,A -85,B 0,C 180,E1 -1732.053,E2 -1732.053} C_VEL
LIN {X 0,Y 580.252,Z 278.208,A -85,B 0,C 180,E1 -1734.715,E2 -1734.715} C_VEL
LIN {X 0,Y 580.242,Z 278.201,A -85,B 0,C 180,E1 -1737.403,E2 -1737.403} C_VEL
LIN {X 0,Y 580.248,Z 278.2,A -85,B 0,C 180,E1 -1739.774,E2 -1739.774} C_VEL
LIN {X 0,Y 580.28,Z 278.198,A -85,B 0,C 180,E1 -1742.201,E2 -1742.201} C_VEL
LIN {X 0,Y 580.28,Z 278.204,A -85,B 0,C 180,E1 -1744.696,E2 -1744.696} C_VEL
LIN {X 0,Y 580.29,Z 278.199,A -85,B 0,C 180,E1 -1747.268,E2 -1747.268} C_VEL
LIN {X 0,Y 580.278,Z 278.197,A -85,B 0,C 180,E1 -1750.269,E2 -1750.269} C_VEL
LIN {X 0,Y 580.26,Z 278.204,A -85,B 0,C 180,E1 -1753.389,E2 -1753.389} C_VEL
LIN {X 0,Y 580.234,Z 278.202,A -85,B 0,C 180,E1 -1756.338,E2 -1756.338} C_VEL
LIN {X 0,Y 580.286,Z 278.205,A -85,B 0,C 180,E1 -1759.156,E2 -1759.156} C_VEL
LIN {X 0,Y 580.28,Z 278.197,A -85,B 0,C 180,E1 -1761.927,E2 -1761.927} C_VEL
LIN {X 0,Y 580.239,Z 278.201,A -85,B 0,C 180,E1 -1764.452,E2 -1764.452} C_VEL
LIN {X 0,Y 580.281,Z 278.199,A -85,B 0,C 180,E1 -1766.975,E2 -1766.975} C_VEL
LIN {X 0,Y 580.285,Z 278.205,A -85,B 0,C 180,E1 -1769.424,E2 -1769.424} C_VEL
LIN {X 0,Y 580.251,Z 278.202,A -85,B 0,C 180,E1 -1772.148,E2 -1772.148} C_VEL
LIN {X 0,Y 580.294,Z 278.195,A -85,B 0,C 180,E1 -1774.92,E2 -1774.92} C_VEL
LIN {X 0,Y 580.263,Z 278.205,A -85,B 0,C 180,E1 -1777.947,E2 -1777.947} C_VEL
LIN {X 0,Y 580.283,Z 278.196,A -85,B 0,C 180,E1 -1780.913,E2 -1780.913} C_VEL
LIN {X 0,Y 580.294,Z 278.195,A -85,B 0,C 180,E1 -1783.102,E2 -1783.102} C_VEL
LIN {X 0,Y 580.306,Z 278.203,A -85,B 0,C 180,E1 -1785.983,E2 -1785.983} C_VEL
LIN {X 0,Y 580.295,Z 278.195,A -85,B 0,C 180,E1 -1788.827,E2 -1788.827} C_VEL
LIN {X 0,Y 580.318,Z 278.195,A -85,B 0,C 180,E1 -1791.644,E2 -1791.644} C_VEL
LIN {X 0,Y 580.322,Z 278.197,A -85,B 0,C 180,E1 -1794.44,E2 -1794.44} C_VEL
LIN {X 0,Y 580.325,Z 278.19,A -85,B 0,C 180,E1 -1797.223,E2 -1797.223} C_VEL
LIN {X 0,Y 580.338,Z 278.194,A -85,B 0,C 180,E1 -1800,E2 -1800} C_VEL
LIN {X 0,Y 580.338,Z 278.193,A -85,B 0,C 180,E1 -1802.777,E2 -1802.777} C_VEL
LIN {X 0,Y 580.315,Z 278.192,A -85,B 0,C 180,E1 -1805.56,E2 -1805.56} C_VEL
LIN {X 0,Y 580.325,Z 278.198,A -85,B 0,C 180,E1 -1808.356,E2 -1808.356} C_VEL
LIN {X 0,Y 580.325,Z 278.192,A -85,B 0,C 180,E1 -1811.209,E2 -1811.209} C_VEL
LIN {X 0,Y 580.306,Z 278.198,A -85,B 0,C 180,E1 -1814.339,E2 -1814.339} C_VEL
LIN {X 0,Y 580.303,Z 278.202,A -85,B 0,C 180,E1 -1816.914,E2 -1816.914} C_VEL
LIN {X 0,Y 580.297,Z 278.194,A -85,B 0,C 180,E1 -1819.823,E2 -1819.823} C_VEL
LIN {X 0,Y 580.288,Z 278.204,A -85,B 0,C 180,E1 -1822.803,E2 -1822.803} C_VEL
LIN {X 0,Y 580.301,Z 278.203,A -85,B 0,C 180,E1 -1825.08,E2 -1825.08} C_VEL
LIN {X 0,Y 580.291,Z 278.195,A -85,B 0,C 180,E1 -1827.86,E2 -1827.86} C_VEL
LIN {X 0,Y 580.293,Z 278.198,A -85,B 0,C 180,E1 -1830.698,E2 -1830.698} C_VEL
LIN {X 0,Y 580.298,Z 278.203,A -85,B 0,C 180,E1 -1833.317,E2 -1833.317} C_VEL
LIN {X 0,Y 580.27,Z 278.2,A -85,B 0,C 180,E1 -1835.761,E2 -1835.761} C_VEL
LIN {X 0,Y 580.284,Z 278.196,A -85,B 0,C 180,E1 -1838.147,E2 -1838.147} C_VEL
LIN {X 0,Y 580.295,Z 278.196,A -85,B 0,C 180,E1 -1840.844,E2 -1840.844} C_VEL
LIN {X 0,Y 580.274,Z 278.204,A -85,B 0,C 180,E1 -1843.659,E2 -1843.659} C_VEL
LIN {X 0,Y 580.273,Z 278.197,A -85,B 0,C 180,E1 -1846.61,E2 -1846.61} C_VEL
LIN {X 0,Y 580.296,Z 278.197,A -85,B 0,C 180,E1 -1849.158,E2 -1849.158} C_VEL
LIN {X 0,Y 580.287,Z 278.202,A -85,B 0,C 180,E1 -1851.928,E2 -1851.928} C_VEL
LIN {X 0,Y 580.249,Z 278.201,A -85,B 0,C 180,E1 -1854.454,E2 -1854.454} C_VEL
LIN {X 0,Y 580.288,Z 278.195,A -85,B 0,C 180,E1 -1856.976,E2 -1856.976} C_VEL
LIN {X 0,Y 580.295,Z 278.197,A -85,B 0,C 180,E1 -1859.426,E2 -1859.426} C_VEL
LIN {X 0,Y 580.298,Z 278.203,A -85,B 0,C 180,E1 -1862.142,E2 -1862.142} C_VEL
LIN {X 0,Y 580.321,Z 278.193,A -85,B 0,C 180,E1 -1865.271,E2 -1865.271} C_VEL
LIN {X 0,Y 580.309,Z 278.275,A -85,B 0,C 180,E1 -1866.659,E2 -1866.659} C_VEL
LIN {X 0,Y 580.973,Z 283.351,A -85,B 0,C 180,E1 -1867.414,E2 -1867.414} C_VEL
LIN {X 0,Y 580.754,Z 305.062,A -85,B 0,C 180,E1 -1870.521,E2 -1870.521} C_VEL
LIN {X 0,Y 580.545,Z 326.068,A -85,B 0,C 180,E1 -1873.472,E2 -1873.472} C_VEL
LIN {X 0,Y 580.398,Z 346.617,A -85,B 0,C 180,E1 -1876.32,E2 -1876.32} C_VEL
LIN {X 0,Y 580.987,Z 352.554,A -85,B 0,C 180,E1 -1876.424,E2 -1876.424} C_VEL
LIN {X 0,Y 580.786,Z 454.975,A -85,B 0,C 180,E1 -1877.708,E2 -1877.708} C_VEL
LIN {X 0,Y 580.729,Z 468.238,A -85,B 0,C 180,E1 -1878.017,E2 -1878.017} C_VEL
LIN {X 0,Y 580.663,Z 480.387,A -85,B 0,C 180,E1 -1878.437,E2 -1878.437} C_VEL
LIN {X 0,Y 580.574,Z 492.638,A -85,B 0,C 180,E1 -1879.009,E2 -1879.009} C_VEL
LIN {X 0,Y 580.421,Z 504.21,A -85,B 0,C 180,E1 -1879.712,E2 -1879.712} C_VEL
LIN {X 0,Y 580.342,Z 514.606,A -85,B 0,C 180,E1 -1880.503,E2 -1880.503} C_VEL
LIN {X 0,Y 580.262,Z 523.061,A -85,B 0,C 180,E1 -1881.293,E2 -1881.293} C_VEL
LIN {X 0,Y 580.221,Z 530.965,A -85,B 0,C 180,E1 -1882.169,E2 -1882.169} C_VEL
LIN {X 0,Y 580.156,Z 538.638,A -85,B 0,C 180,E1 -1883.22,E2 -1883.22} C_VEL
LIN {X 0,Y 580.139,Z 545.682,A -85,B 0,C 180,E1 -1884.439,E2 -1884.439} C_VEL
LIN {X 0,Y 580.108,Z 550.374,A -85,B 0,C 180,E1 -1885.484,E2 -1885.484} C_VEL
LIN {X 0,Y 580.122,Z 553.958,A -85,B 0,C 180,E1 -1886.528,E2 -1886.528} C_VEL
LIN {X 0,Y 580.043,Z 555.809,A -85,B 0,C 180,E1 -1887.222,E2 -1887.222} C_VEL
LIN {X 0,Y 580.038,Z 557.2,A -85,B 0,C 180,E1 -1887.917,E2 -1887.917} C_VEL
LIN {X 0,Y 580.04,Z 558.785,A -85,B 0,C 180,E1 -1889.306,E2 -1889.306} C_VEL
LIN {X 0,Y 580.037,Z 559,A -85,B 0,C 180,E1 -1890,E2 -1890} C_VEL
LIN {X 0,Y 580.046,Z 558.186,A -85,B 0,C 180,E1 -1891.389,E2 -1891.389} C_VEL
LIN {X 0,Y 580.038,Z 557.199,A -85,B 0,C 180,E1 -1892.083,E2 -1892.083} C_VEL
LIN {X 0,Y 580.043,Z 555.809,A -85,B 0,C 180,E1 -1892.778,E2 -1892.778} C_VEL
LIN {X 0,Y 580.109,Z 552.895,A -85,B 0,C 180,E1 -1893.821,E2 -1893.821} C_VEL
LIN {X 0,Y 580.053,Z 548.948,A -85,B 0,C 180,E1 -1894.866,E2 -1894.866} C_VEL
LIN {X 0,Y 580.14,Z 542.875,A -85,B 0,C 180,E1 -1896.085,E2 -1896.085} C_VEL
LIN {X 0,Y 580.184,Z 536.235,A -85,B 0,C 180,E1 -1897.133,E2 -1897.133} C_VEL
LIN {X 0,Y 580.246,Z 527.988,A -85,B 0,C 180,E1 -1898.182,E2 -1898.182} C_VEL
LIN {X 0,Y 580.333,Z 517.599,A -85,B 0,C 180,E1 -1899.234,E2 -1899.234} C_VEL
LIN {X 0,Y 580.43,Z 507.923,A -85,B 0,C 180,E1 -1900.024,E2 -1900.024} C_VEL
LIN {X 0,Y 580.531,Z 497.323,A -85,B 0,C 180,E1 -1900.727,E2 -1900.727} C_VEL
LIN {X 0,Y 580.613,Z 485.482,A -85,B 0,C 180,E1 -1901.344,E2 -1901.344} C_VEL
LIN {X 0,Y 580.653,Z 473.167,A -85,B 0,C 180,E1 -1901.83,E2 -1901.83} C_VEL
LIN {X 0,Y 580.755,Z 460.511,A -85,B 0,C 180,E1 -1902.182,E2 -1902.182} C_VEL
LIN {X 0,Y 580.835,Z 447.293,A -85,B 0,C 180,E1 -1902.402,E2 -1902.402} C_VEL
LIN {X 0,Y 580.805,Z 349.364,A -85,B 0,C 180,E1 -1903.62,E2 -1903.62} C_VEL
LIN {X 0,Y 580.398,Z 346.611,A -85,B 0,C 180,E1 -1903.68,E2 -1903.68} C_VEL
LIN {X 0,Y 580.545,Z 326.062,A -85,B 0,C 180,E1 -1906.528,E2 -1906.528} C_VEL
LIN {X 0,Y 580.754,Z 305.063,A -85,B 0,C 180,E1 -1909.479,E2 -1909.479} C_VEL
LIN {X 0,Y 580.964,Z 284.64,A -85,B 0,C 180,E1 -1912.399,E2 -1912.399} C_VEL
LIN {X 0,Y 580.635,Z 279.955,A -85,B 0,C 180,E1 -1913.088,E2 -1913.088} C_VEL
LIN {X 0,Y 580.312,Z 278.201,A -85,B 0,C 180,E1 -1913.377,E2 -1913.377} C_VEL
LIN {X 0,Y 580.279,Z 278.207,A -85,B 0,C 180,E1 -1915.85,E2 -1915.85} C_VEL
LIN {X 0,Y 580.298,Z 278.204,A -85,B 0,C 180,E1 -1918.186,E2 -1918.186} C_VEL
LIN {X 0,Y 580.286,Z 278.199,A -85,B 0,C 180,E1 -1920.694,E2 -1920.694} C_VEL
LIN {X 0,Y 580.285,Z 278.196,A -85,B 0,C 180,E1 -1923.313,E2 -1923.313} C_VEL
LIN {X 0,Y 580.246,Z 278.203,A -85,B 0,C 180,E1 -1925.756,E2 -1925.756} C_VEL
LIN {X 0,Y 580.288,Z 278.202,A -85,B 0,C 180,E1 -1928.146,E2 -1928.146} C_VEL
LIN {X 0,Y 580.298,Z 278.199,A -85,B 0,C 180,E1 -1930.843,E2 -1930.843} C_VEL
LIN {X 0,Y 580.273,Z 278.197,A -85,B 0,C 180,E1 -1933.658,E2 -1933.658} C_VEL
LIN {X 0,Y 580.275,Z 278.208,A -85,B 0,C 180,E1 -1936.609,E2 -1936.609} C_VEL
LIN {X 0,Y 580.298,Z 278.197,A -85,B 0,C 180,E1 -1939.156,E2 -1939.156} C_VEL
LIN {X 0,Y 580.29,Z 278.195,A -85,B 0,C 180,E1 -1941.927,E2 -1941.927} C_VEL
LIN {X 0,Y 580.25,Z 278.203,A -85,B 0,C 180,E1 -1944.452,E2 -1944.452} C_VEL
LIN {X 0,Y 580.288,Z 278.206,A -85,B 0,C 180,E1 -1946.975,E2 -1946.975} C_VEL
LIN {X 0,Y 580.295,Z 278.198,A -85,B 0,C 180,E1 -1949.425,E2 -1949.425} C_VEL
LIN {X 0,Y 580.296,Z 278.194,A -85,B 0,C 180,E1 -1952.141,E2 -1952.141} C_VEL
LIN {X 0,Y 580.32,Z 278.202,A -85,B 0,C 180,E1 -1955.269,E2 -1955.269} C_VEL
LIN {X 0,Y 580.27,Z 278.199,A -85,B 0,C 180,E1 -1957.947,E2 -1957.947} C_VEL
LIN {X 0,Y 580.317,Z 278.194,A -85,B 0,C 180,E1 -1960.914,E2 -1960.914} C_VEL
LIN {X 0,Y 580.276,Z 278.201,A -85,B 0,C 180,E1 -1963.825,E2 -1963.825} C_VEL
LIN {X 0,Y 580.323,Z 278.194,A -85,B 0,C 180,E1 -1965.983,E2 -1965.983} C_VEL
LIN {X 0,Y 580.302,Z 278.193,A -85,B 0,C 180,E1 -1968.827,E2 -1968.827} C_VEL
LIN {X 0,Y 580.325,Z 278.199,A -85,B 0,C 180,E1 -1971.644,E2 -1971.644} C_VEL
LIN {X 0,Y 580.322,Z 278.191,A -85,B 0,C 180,E1 -1974.44,E2 -1974.44} C_VEL
LIN {X 0,Y 580.334,Z 278.19,A -85,B 0,C 180,E1 -1977.223,E2 -1977.223} C_VEL
LIN {X 0,Y 580.351,Z 278.197,A -85,B 0,C 180,E1 -1980,E2 -1980} C_VEL
LIN {X 0,Y 580.335,Z 278.189,A -85,B 0,C 180,E1 -1982.776,E2 -1982.776} C_VEL
LIN {X 0,Y 580.322,Z 278.192,A -85,B 0,C 180,E1 -1985.56,E2 -1985.56} C_VEL
LIN {X 0,Y 580.325,Z 278.2,A -85,B 0,C 180,E1 -1988.356,E2 -1988.356} C_VEL
LIN {X 0,Y 580.297,Z 278.194,A -85,B 0,C 180,E1 -1991.191,E2 -1991.191} C_VEL
LIN {X 0,Y 580.323,Z 278.194,A -85,B 0,C 180,E1 -1994.017,E2 -1994.017} C_VEL
LIN {X 0,Y 580.31,Z 278.197,A -85,B 0,C 180,E1 -1996.914,E2 -1996.914} C_VEL
LIN {X 0,Y 580.302,Z 278.194,A -85,B 0,C 180,E1 -1999.822,E2 -1999.822} C_VEL
LIN {X 0,Y 580.281,Z 278.197,A -85,B 0,C 180,E1 -2001.325,E2 -2001.325} C_VEL
LIN {X 0,Y 579.583,Z 278.285,A -85,B 0,C 180,E1 -2001.905,E2 -2001.905} C_VEL
LIN {X 0,Y 576.707,Z 278.65,A -85,B 0,C 180,E1 -2002.845,E2 -2002.845} C_VEL
LIN {X 0,Y 574.313,Z 278.943,A -85,B 0,C 180,E1 -2003.601,E2 -2003.601} C_VEL
LIN {X 0,Y 573.314,Z 279.066,A -85,B 0,C 180,E1 -2004.185,E2 -2004.185} C_VEL
LIN {X 0,Y 573.248,Z 279.076,A -85,B 0,C 180,E1 -2004.382,E2 -2004.382} C_VEL
LIN {X 0,Y 573.249,Z 279.08,A -85,B 0,C 180,E1 -2006.976,E2 -2006.976} C_VEL
LIN {X 0,Y 573.245,Z 279.075,A -85,B 0,C 180,E1 -2009.488,E2 -2009.488} C_VEL
LIN {X 0,Y 573.251,Z 279.075,A -85,B 0,C 180,E1 -2012.645,E2 -2012.645} C_VEL
LIN {X 0,Y 573.205,Z 279.087,A -85,B 0,C 180,E1 -2015.188,E2 -2015.188} C_VEL
LIN {X 0,Y 573.234,Z 279.075,A -85,B 0,C 180,E1 -2017.808,E2 -2017.808} C_VEL
LIN {X 0,Y 573.243,Z 279.073,A -85,B 0,C 180,E1 -2020.525,E2 -2020.525} C_VEL
LIN {X 0,Y 573.237,Z 279.084,A -85,B 0,C 180,E1 -2023.359,E2 -2023.359} C_VEL
LIN {X 0,Y 573.236,Z 279.074,A -85,B 0,C 180,E1 -2026.641,E2 -2026.641} C_VEL
LIN {X 0,Y 573.244,Z 279.082,A -85,B 0,C 180,E1 -2029.475,E2 -2029.475} C_VEL
LIN {X 0,Y 573.235,Z 279.077,A -85,B 0,C 180,E1 -2032.193,E2 -2032.193} C_VEL
LIN {X 0,Y 573.233,Z 279.077,A -85,B 0,C 180,E1 -2035.229,E2 -2035.229} C_VEL
LIN {X 0,Y 573.251,Z 279.083,A -85,B 0,C 180,E1 -2037.772,E2 -2037.772} C_VEL
LIN {X 0,Y 573.306,Z 279.143,A -85,B 0,C 180,E1 -2040.938,E2 -2040.938} C_VEL
LIN {X 0,Y 573.408,Z 287.348,A -85,B 0,C 180,E1 -2042.44,E2 -2042.44} C_VEL
LIN {X 0,Y 573.31,Z 304.673,A -85,B 0,C 180,E1 -2045.561,E2 -2045.561} C_VEL
LIN {X 0,Y 573.226,Z 308.384,A -85,B 0,C 180,E1 -2046.222,E2 -2046.222} C_VEL
LIN {X 0,Y 574.1,Z 314.561,A -85,B 0,C 180,E1 -2046.328,E2 -2046.328} C_VEL
LIN {X 0,Y 573.803,Z 415.632,A -85,B 0,C 180,E1 -2047.614,E2 -2047.614} C_VEL
LIN {X 0,Y 573.71,Z 429.202,A -85,B 0,C 180,E1 -2047.942,E2 -2047.942} C_VEL
LIN {X 0,Y 573.666,Z 441.64,A -85,B 0,C 180,E1 -2048.389,E2 -2048.389} C_VEL
LIN {X 0,Y 573.546,Z 453.399,A -85,B 0,C 180,E1 -2048.961,E2 -2048.961} C_VEL
LIN {X 0,Y 573.406,Z 464.471,A -85,B 0,C 180,E1 -2049.648,E2 -2049.648} C_VEL
LIN {X 0,Y 573.326,Z 475.259,A -85,B 0,C 180,E1 -2050.486,E2 -2050.486} C_VEL
LIN {X 0,Y 573.246,Z 484.815,A -85,B 0,C 180,E1 -2051.412,E2 -2051.412} C_VEL
LIN {X 0,Y 573.133,Z 492.635,A -85,B 0,C 180,E1 -2052.332,E2 -2052.332} C_VEL
LIN {X 0,Y 573.101,Z 499.568,A -85,B 0,C 180,E1 -2053.328,E2 -2053.328} C_VEL
LIN {X 0,Y 573.027,Z 505.331,A -85,B 0,C 180,E1 -2054.346,E2 -2054.346} C_VEL
LIN {X 0,Y 573.015,Z 510.205,A -85,B 0,C 180,E1 -2055.431,E2 -2055.431} C_VEL
LIN {X 0,Y 573.003,Z 513.943,A -85,B 0,C 180,E1 -2056.524,E2 -2056.524} C_VEL
LIN {X 0,Y 572.955,Z 515.837,A -85,B 0,C 180,E1 -2057.244,E2 -2057.244} C_VEL
LIN {X 0,Y 572.948,Z 517.243,A -85,B 0,C 180,E1 -2057.964,E2 -2057.964} C_VEL
LIN {X 0,Y 572.984,Z 518.461,A -85,B 0,C 180,E1 -2058.887,E2 -2058.887} C_VEL
LIN {X 0,Y 572.974,Z 518.991,A -85,B 0,C 180,E1 -2060.112,E2 -2060.112} C_VEL
LIN {X 0,Y 572.949,Z 518.089,A -85,B 0,C 180,E1 -2061.535,E2 -2061.535} C_VEL
LIN {X 0,Y 572.976,Z 517.051,A -85,B 0,C 180,E1 -2062.246,E2 -2062.246} C_VEL
LIN {X 0,Y 573.029,Z 514.342,A -85,B 0,C 180,E1 -2063.432,E2 -2063.432} C_VEL
LIN {X 0,Y 572.996,Z 509.954,A -85,B 0,C 180,E1 -2064.722,E2 -2064.722} C_VEL
LIN {X 0,Y 573.035,Z 505.147,A -85,B 0,C 180,E1 -2065.78,E2 -2065.78} C_VEL
LIN {X 0,Y 573.057,Z 499.105,A -85,B 0,C 180,E1 -2066.836,E2 -2066.836} C_VEL
LIN {X 0,Y 573.114,Z 491.613,A -85,B 0,C 180,E1 -2067.891,E2 -2067.891} C_VEL
LIN {X 0,Y 573.241,Z 483.934,A -85,B 0,C 180,E1 -2068.77,E2 -2068.77} C_VEL
LIN {X 0,Y 573.3,Z 474.739,A -85,B 0,C 180,E1 -2069.648,E2 -2069.648} C_VEL
LIN {X 0,Y 573.39,Z 464.521,A -85,B 0,C 180,E1 -2070.439,E2 -2070.439} C_VEL
LIN {X 0,Y 573.558,Z 453.189,A -85,B 0,C 180,E1 -2071.141,E2 -2071.141} C_VEL
LIN {X 0,Y 573.694,Z 441.387,A -85,B 0,C 180,E1 -2071.711,E2 -2071.711} C_VEL
LIN {X 0,Y 573.742,Z 428.386,A -85,B 0,C 180,E1 -2072.171,E2 -2072.171} C_VEL
LIN {X 0,Y 573.847,Z 415.455,A -85,B 0,C 180,E1 -2072.478,E2 -2072.478} C_VEL
LIN {X 0,Y 573.968,Z 312.977,A -85,B 0,C 180,E1 -2073.785,E2 -2073.785} C_VEL
LIN {X 0,Y 573.234,Z 308.396,A -85,B 0,C 180,E1 -2073.866,E2 -2073.866} C_VEL
LIN {X 0,Y 573.389,Z 294.626,A -85,B 0,C 180,E1 -2076.333,E2 -2076.333} C_VEL
LIN {X 0,Y 573.435,Z 280.974,A -85,B 0,C 180,E1 -2078.812,E2 -2078.812} C_VEL
LIN {X 0,Y 573.224,Z 279.081,A -85,B 0,C 180,E1 -2079.171,E2 -2079.171} C_VEL
LIN {X 0,Y 573.23,Z 279.083,A -85,B 0,C 180,E1 -2082.03,E2 -2082.03} C_VEL
LIN {X 0,Y 573.221,Z 279.077,A -85,B 0,C 180,E1 -2084.919,E2 -2084.919} C_VEL
LIN {X 0,Y 573.208,Z 279.079,A -85,B 0,C 180,E1 -2087.849,E2 -2087.849} C_VEL
LIN {X 0,Y 573.246,Z 279.077,A -85,B 0,C 180,E1 -2090.826,E2 -2090.826} C_VEL
LIN {X 0,Y 573.21,Z 279.078,A -85,B 0,C 180,E1 -2093.138,E2 -2093.138} C_VEL
LIN {X 0,Y 573.199,Z 279.078,A -85,B 0,C 180,E1 -2095.412,E2 -2095.412} C_VEL
LIN {X 0,Y 573.2,Z 279.079,A -85,B 0,C 180,E1 -2098.019,E2 -2098.019} C_VEL
LIN {X 0,Y 573.215,Z 279.078,A -85,B 0,C 180,E1 -2100.177,E2 -2100.177} C_VEL
LIN {X 0,Y 573.241,Z 279.081,A -85,B 0,C 180,E1 -2102.645,E2 -2102.645} C_VEL
LIN {X 0,Y 573.199,Z 279.083,A -85,B 0,C 180,E1 -2105.187,E2 -2105.187} C_VEL
LIN {X 0,Y 573.224,Z 279.075,A -85,B 0,C 180,E1 -2107.807,E2 -2107.807} C_VEL
LIN {X 0,Y 573.239,Z 279.076,A -85,B 0,C 180,E1 -2110.524,E2 -2110.524} C_VEL
LIN {X 0,Y 573.229,Z 279.076,A -85,B 0,C 180,E1 -2113.667,E2 -2113.667} C_VEL
LIN {X 0,Y 573.202,Z 279.08,A -85,B 0,C 180,E1 -2116.637,E2 -2116.637} C_VEL
LIN {X 0,Y 573.238,Z 279.08,A -85,B 0,C 180,E1 -2119.474,E2 -2119.474} C_VEL
LIN {X 0,Y 573.226,Z 279.075,A -85,B 0,C 180,E1 -2122.192,E2 -2122.192} C_VEL
LIN {X 0,Y 573.224,Z 279.083,A -85,B 0,C 180,E1 -2125.229,E2 -2125.229} C_VEL
LIN {X 0,Y 573.243,Z 279.078,A -85,B 0,C 180,E1 -2127.771,E2 -2127.771} C_VEL
LIN {X 0,Y 573.252,Z 279.072,A -85,B 0,C 180,E1 -2130.633,E2 -2130.633} C_VEL
LIN {X 0,Y 573.254,Z 279.079,A -85,B 0,C 180,E1 -2133.81,E2 -2133.81} C_VEL
LIN {X 0,Y 573.219,Z 279.079,A -85,B 0,C 180,E1 -2136.134,E2 -2136.134} C_VEL
LIN {X 0,Y 573.24,Z 279.075,A -85,B 0,C 180,E1 -2139.173,E2 -2139.173} C_VEL
LIN {X 0,Y 573.216,Z 279.08,A -85,B 0,C 180,E1 -2141.411,E2 -2141.411} C_VEL
LIN {X 0,Y 573.237,Z 279.08,A -85,B 0,C 180,E1 -2143.621,E2 -2143.621} C_VEL
LIN {X 0,Y 573.218,Z 279.078,A -85,B 0,C 180,E1 -2146.529,E2 -2146.529} C_VEL
LIN {X 0,Y 573.253,Z 279.072,A -85,B 0,C 180,E1 -2148.745,E2 -2148.745} C_VEL
LIN {X 0,Y 573.274,Z 279.071,A -85,B 0,C 180,E1 -2151.54,E2 -2151.54} C_VEL
LIN {X 0,Y 573.287,Z 279.074,A -85,B 0,C 180,E1 -2154.372,E2 -2154.372} C_VEL
LIN {X 0,Y 573.293,Z 279.066,A -85,B 0,C 180,E1 -2157.189,E2 -2157.189} C_VEL
LIN {X 0,Y 573.308,Z 279.07,A -85,B 0,C 180,E1 -2160,E2 -2160} C_VEL
LIN {X 0,Y 573.303,Z 279.069,A -85,B 0,C 180,E1 -2162.811,E2 -2162.811} C_VEL
LIN {X 0,Y 573.281,Z 279.068,A -85,B 0,C 180,E1 -2165.628,E2 -2165.628} C_VEL
LIN {X 0,Y 573.297,Z 279.076,A -85,B 0,C 180,E1 -2168.459,E2 -2168.459} C_VEL
LIN {X 0,Y 573.291,Z 279.068,A -85,B 0,C 180,E1 -2171.312,E2 -2171.312} C_VEL
LIN {X 0,Y 573.272,Z 279.075,A -85,B 0,C 180,E1 -2174.425,E2 -2174.425} C_VEL
LIN {X 0,Y 573.25,Z 279.077,A -85,B 0,C 180,E1 -2177.112,E2 -2177.112} C_VEL
LIN {X 0,Y 573.244,Z 279.073,A -85,B 0,C 180,E1 -2180.077,E2 -2180.077} C_VEL
LIN {X 0,Y 573.226,Z 279.083,A -85,B 0,C 180,E1 -2183.1,E2 -2183.1} C_VEL
LIN {X 0,Y 573.249,Z 279.076,A -85,B 0,C 180,E1 -2185.41,E2 -2185.41} C_VEL
LIN {X 0,Y 573.245,Z 279.072,A -85,B 0,C 180,E1 -2188.03,E2 -2188.03} C_VEL
LIN {X 0,Y 573.237,Z 279.08,A -85,B 0,C 180,E1 -2190.886,E2 -2190.886} C_VEL
LIN {X 0,Y 573.256,Z 279.076,A -85,B 0,C 180,E1 -2193.525,E2 -2193.525} C_VEL
LIN {X 0,Y 573.239,Z 279.074,A -85,B 0,C 180,E1 -2196.05,E2 -2196.05} C_VEL
LIN {X 0,Y 573.243,Z 279.074,A -85,B 0,C 180,E1 -2198.702,E2 -2198.702} C_VEL
LIN {X 0,Y 573.249,Z 279.08,A -85,B 0,C 180,E1 -2201.596,E2 -2201.596} C_VEL
LIN {X 0,Y 573.231,Z 279.074,A -85,B 0,C 180,E1 -2204.334,E2 -2204.334} C_VEL
LIN {X 0,Y 573.237,Z 279.08,A -85,B 0,C 180,E1 -2207.359,E2 -2207.359} C_VEL
LIN {X 0,Y 573.236,Z 279.074,A -85,B 0,C 180,E1 -2210.393,E2 -2210.393} C_VEL
LIN {X 0,Y 573.25,Z 279.073,A -85,B 0,C 180,E1 -2213.078,E2 -2213.078} C_VEL
LIN {X 0,Y 573.265,Z 279.079,A -85,B 0,C 180,E1 -2215.672,E2 -2215.672} C_VEL
LIN {X 0,Y 573.239,Z 279.078,A -85,B 0,C 180,E1 -2218.185,E2 -2218.185} C_VEL
LIN {X 0,Y 573.263,Z 279.072,A -85,B 0,C 180,E1 -2220.635,E2 -2220.635} C_VEL
LIN {X 0,Y 573.25,Z 279.073,A -85,B 0,C 180,E1 -2223.025,E2 -2223.025} C_VEL
LIN {X 0,Y 573.275,Z 279.072,A -85,B 0,C 180,E1 -2225.367,E2 -2225.367} C_VEL
LIN {X 0,Y 573.277,Z 279.211,A -85,B 0,C 180,E1 -2226.528,E2 -2226.528} C_VEL
LIN {X 0,Y 574.049,Z 284.465,A -85,B 0,C 180,E1 -2227.317,E2 -2227.317} C_VEL
LIN {X 0,Y 573.807,Z 305.359,A -85,B 0,C 180,E1 -2230.318,E2 -2230.318} C_VEL
LIN {X 0,Y 573.568,Z 326.123,A -85,B 0,C 180,E1 -2233.273,E2 -2233.273} C_VEL
LIN {X 0,Y 573.392,Z 346.617,A -85,B 0,C 180,E1 -2236.15,E2 -2236.15} C_VEL
LIN {X 0,Y 574.1,Z 352.554,A -85,B 0,C 180,E1 -2236.258,E2 -2236.258} C_VEL
LIN {X 0,Y 573.866,Z 454.975,A -85,B 0,C 180,E1 -2237.558,E2 -2237.558} C_VEL
LIN {X 0,Y 573.788,Z 468.237,A -85,B 0,C 180,E1 -2237.87,E2 -2237.87} C_VEL
LIN {X 0,Y 573.691,Z 480.389,A -85,B 0,C 180,E1 -2238.294,E2 -2238.294} C_VEL
LIN {X 0,Y 573.588,Z 492.643,A -85,B 0,C 180,E1 -2238.874,E2 -2238.874} C_VEL
LIN {X 0,Y 573.437,Z 504.208,A -85,B 0,C 180,E1 -2239.586,E2 -2239.586} C_VEL
LIN {X 0,Y 573.328,Z 514.607,A -85,B 0,C 180,E1 -2240.386,E2 -2240.386} C_VEL
LIN {X 0,Y 573.237,Z 523.074,A -85,B 0,C 180,E1 -2241.185,E2 -2241.185} C_VEL
LIN {X 0,Y 573.16,Z 530.965,A -85,B 0,C 180,E1 -2242.071,E2 -2242.071} C_VEL
LIN {X 0,Y 573.074,Z 538.943,A -85,B 0,C 180,E1 -2243.184,E2 -2243.184} C_VEL
LIN {X 0,Y 573.07,Z 545.682,A -85,B 0,C 180,E1 -2244.37,E2 -2244.37} C_VEL
LIN {X 0,Y 573.028,Z 550.374,A -85,B 0,C 180,E1 -2245.428,E2 -2245.428} C_VEL
LIN {X 0,Y 573.022,Z 553.959,A -85,B 0,C 180,E1 -2246.485,E2 -2246.485} C_VEL
LIN {X 0,Y 572.959,Z 555.809,A -85,B 0,C 180,E1 -2247.188,E2 -2247.188} C_VEL
LIN {X 0,Y 572.946,Z 558.186,A -85,B 0,C 180,E1 -2248.595,E2 -2248.595} C_VEL
LIN {X 0,Y 572.938,Z 559,A -85,B 0,C 180,E1 -2250,E2 -2250} C_VEL
LIN {X 0,Y 572.946,Z 558.186,A -85,B 0,C 180,E1 -2251.406,E2 -2251.406} C_VEL
LIN {X 0,Y 572.938,Z 557.199,A -85,B 0,C 180,E1 -2252.109,E2 -2252.109} C_VEL
LIN {X 0,Y 572.959,Z 555.809,A -85,B 0,C 180,E1 -2252.813,E2 -2252.813} C_VEL
